KUKA KRL program: MyProgram_121().src

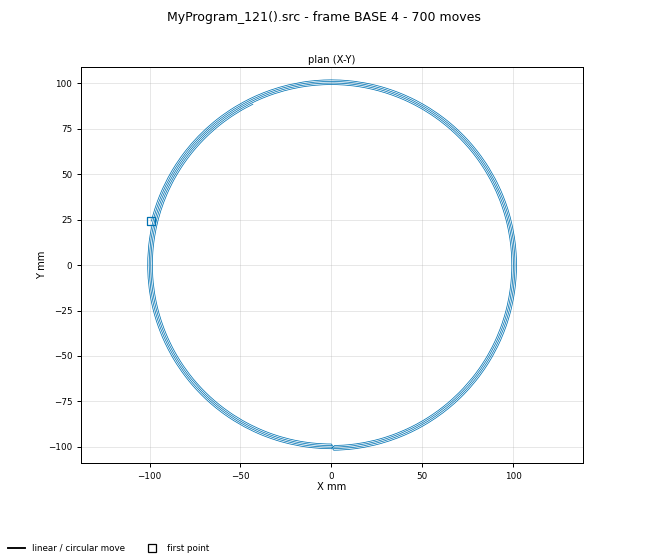
[picture p0: tool path of MyProgram_121().src in frame BASE 4, 700 of 700 moves have a stored position in this frame; points joined in program order, loops and branches not executed]
&ACCESS RVP
&REL 1
&PARAM TEMPLATE = C:\KRC\Roboter\Template\vorgabe
&PARAM EDITMASK = *
DEF MyProgram_121()
; ---- Setting reference (Base) ----
$BASE = BASE_DATA[4]

; --------------------------
; ---- Setting tool (TCP) ----
$TOOL = TOOL_DATA[3]
; --------------------------

$VEL.CP = VEL_APROX_PRINT
Startdeposition()
$VEL.CP = VEL_PRINT
LIN {X -98.957,Y 24.1948,Z 102,A 161.3136,B 24.9312,C -1.9162,E1 24.8447,E2 -75.7869} C_DIS
LIN {X -98.1679,Y 27.2258,Z 102,A 159.187,B 24.9317,C -1.9094,E1 24.8462,E2 -73.6317} C_DIS
LIN {X -97.1085,Y 30.7923,Z 102,A 156.6963,B 24.9321,C -1.9025,E1 24.8484,E2 -71.1104} C_DIS
LIN {X -95.7541,Y 34.7715,Z 102,A 155.0992,B 24.9297,C -1.9358,E1 24.8498,E2 -69.5835} C_DIS
LIN {X -94.7978,Y 37.2995,Z 102,A 153.5612,B 24.9294,C -1.9399,E1 24.8513,E2 -68.0466} C_DIS
LIN {X -93.6877,Y 40.0091,Z 102,A 151.9205,B 24.9291,C -1.9451,E1 24.8531,E2 -66.4092} C_DIS
LIN {X -92.7094,Y 42.2256,Z 102,A 150.3541,B 24.9293,C -1.9423,E1 24.8549,E2 -64.8275} C_DIS
LIN {X -89.881,Y 47.9536,Z 102,A 146.8815,B 24.9282,C -1.957,E1 24.8593,E2 -61.3714} C_DIS
LIN {X -87.5821,Y 52.0317,Z 102,A 144.2252,B 24.9277,C -1.9639,E1 24.8629,E2 -58.7175} C_DIS
LIN {X -85.5843,Y 55.2562,Z 102,A 141.634,B 24.9284,C -1.9543,E1 24.8668,E2 -56.0904} C_DIS
LIN {X -82.7794,Y 59.3759,Z 102,A 138.6498,B 24.9283,C -1.9558,E1 24.8717,E2 -53.0952} C_DIS
LIN {X -80.5027,Y 62.4283,Z 102,A 137.1356,B 24.9263,C -1.983,E1 24.8741,E2 -51.6386} C_DIS
LIN {X -76.9267,Y 66.7851,Z 102,A 134.0827,B 24.9254,C -1.9953,E1 24.8796,E2 -48.6009} C_DIS
LIN {X -73.2959,Y 70.7502,Z 102,A 130.9039,B 24.9252,C -1.9975,E1 24.8856,E2 -45.4133} C_DIS
LIN {X -69.1212,Y 74.8347,Z 102,A 127.7767,B 24.9242,C -2.0107,E1 24.8919,E2 -42.3047} C_DIS
LIN {X -64.7279,Y 78.6665,Z 102,A 124.3462,B 24.924,C -2.0128,E1 24.8991,E2 -38.8656} C_DIS
LIN {X -62.3244,Y 80.5828,Z 102,A 122.4933,B 24.924,C -2.0122,E1 24.9032,E2 -37.0044} C_DIS
LIN {X -60.1036,Y 82.2523,Z 102,A 120.9648,B 24.9237,C -2.0166,E1 24.9066,E2 -35.481} C_DIS
LIN {X -55.7725,Y 85.2492,Z 102,A 117.9876,B 24.9233,C -2.0219,E1 24.9135,E2 -32.5065} C_DIS
LIN {X -52.8849,Y 87.0693,Z 102,A 115.7015,B 24.924,C -2.0126,E1 24.919,E2 -30.1912} C_DIS
LIN {X -48.0016,Y 89.8555,Z 102,A 112.9772,B 24.9225,C -2.0335,E1 24.9255,E2 -27.5088} C_DIS
LIN {X -44.7125,Y 91.5369,Z 102,A 110.1519,B 24.9242,C -2.0105,E1 24.9327,E2 -24.6211} C_DIS
LIN {X -41.1942,Y 93.1711,Z 102,A 108.2639,B 24.9232,C -2.0241,E1 24.9375,E2 -22.761} C_DIS
LIN {X -37.1448,Y 94.8586,Z 102,A 106.1045,B 24.9221,C -2.0385,E1 24.943,E2 -20.631} C_DIS
LIN {X -33.5819,Y 96.1777,Z 102,A 103.6281,B 24.9228,C -2.0291,E1 24.9496,E2 -18.1274} C_DIS
LIN {X -28.5827,Y 97.7807,Z 102,A 101.0832,B 24.9214,C -2.0471,E1 24.9563,E2 -15.6207} C_DIS
LIN {X -23.5966,Y 99.1014,Z 102,A 97.8662,B 24.9221,C -2.0385,E1 24.965,E2 -12.3788} C_DIS
LIN {X -15.5786,Y 100.6736,Z 102,A 93.5985,B 24.9209,C -2.054,E1 24.9767,E2 -8.1433} C_DIS
LIN {X -12.7503,Y 101.0714,Z 102,A 91.1239,B 24.9232,C -2.0235,E1 24.9837,E2 -5.5944} C_DIS
LIN {X -8.267,Y 101.536,Z 102,A 89.0167,B 24.922,C -2.0402,E1 24.9895,E2 -3.5259} C_DIS
LIN {X -4.0963,Y 101.7898,Z 102,A 86.8934,B 24.9212,C -2.0493,E1 24.9953,E2 -1.4237} C_DIS
LIN {X -0.0604,Y 101.8734,Z 102,A 84.4498,B 24.9217,C -2.0434,E1 25.0022,E2 1.0339} C_DIS
LIN {X 4.8959,Y 101.7555,Z 102,A 81.9704,B 24.9208,C -2.0551,E1 25.009,E2 3.4849} C_DIS
LIN {X 8.4387,Y 101.5222,Z 102,A 79.9611,B 24.9208,C -2.0546,E1 25.0146,E2 5.4945} C_DIS
LIN {X 12.6527,Y 101.084,Z 102,A 77.4932,B 24.9211,C -2.051,E1 25.0215,E2 7.9692} C_DIS
LIN {X 18.3069,Y 100.2138,Z 102,A 74.5122,B 24.9205,C -2.0589,E1 25.0297,E2 10.9286} C_DIS
LIN {X 20.8892,Y 99.708,Z 102,A 72.5597,B 24.9219,C -2.0404,E1 25.0351,E2 12.9225} C_DIS
LIN {X 24.06,Y 98.9899,Z 102,A 70.5801,B 24.9224,C -2.0337,E1 25.0405,E2 14.9151} C_DIS
LIN {X 27.3534,Y 98.1318,Z 102,A 69.3081,B 24.9207,C -2.0567,E1 25.0438,E2 16.1306} C_DIS
LIN {X 29.7903,Y 97.4195,Z 102,A 67.1031,B 24.923,C -2.0262,E1 25.0499,E2 18.4039} C_DIS
LIN {X 33.4482,Y 96.2241,Z 102,A 65.5129,B 24.9215,C -2.0461,E1 25.0539,E2 19.9437} C_DIS
LIN {X 36.8556,Y 94.9721,Z 102,A 63.4452,B 24.9217,C -2.0432,E1 25.0593,E2 22.014} C_DIS
LIN {X 39.9474,Y 93.7137,Z 102,A 60.8845,B 24.9239,C -2.0151,E1 25.0661,E2 24.6351} C_DIS
LIN {X 43.9838,Y 91.8875,Z 102,A 59.4721,B 24.9209,C -2.0535,E1 25.0694,E2 25.9529} C_DIS
LIN {X 46.2574,Y 90.7642,Z 102,A 56.8281,B 24.9246,C -2.0049,E1 25.0763,E2 28.7047} C_DIS
LIN {X 50.6903,Y 88.365,Z 102,A 54.8585,B 24.9224,C -2.0341,E1 25.0809,E2 30.5994} C_DIS
LIN {X 54.1717,Y 86.2749,Z 102,A 52.6742,B 24.9224,C -2.0345,E1 25.0861,E2 32.7759} C_DIS
LIN {X 58.6838,Y 83.2733,Z 102,A 49.6805,B 24.9226,C -2.0316,E1 25.093,E2 35.7664} C_DIS
LIN {X 62.2919,Y 80.6078,Z 102,A 46.5734,B 24.9247,C -2.0044,E1 25.1,E2 38.9267} C_DIS
LIN {X 65.02,Y 78.4237,Z 102,A 45.1697,B 24.9233,C -2.0226,E1 25.103,E2 40.2819} C_DIS
LIN {X 67.3026,Y 76.4747,Z 102,A 43.2946,B 24.9241,C -2.0119,E1 25.1069,E2 42.1748} C_DIS
LIN {X 70.2619,Y 73.7665,Z 102,A 41.0725,B 24.9243,C -2.0086,E1 25.1115,E2 44.3956} C_DIS
LIN {X 72.8301,Y 71.2314,Z 102,A 38.6497,B 24.9258,C -1.9888,E1 25.1163,E2 46.8551} C_DIS
LIN {X 75.2471,Y 68.6719,Z 102,A 37.241,B 24.9245,C -2.007,E1 25.1189,E2 48.2146} C_DIS
LIN {X 77.6522,Y 65.9396,Z 102,A 35.1787,B 24.9249,C -2.0017,E1 25.1227,E2 50.2801} C_DIS
LIN {X 80.2578,Y 62.7425,Z 102,A 32.7459,B 24.9256,C -1.9916,E1 25.1269,E2 52.7253} C_DIS
LIN {X 82.4053,Y 59.8946,Z 102,A 30.0003,B 24.9282,C -1.9573,E1 25.1316,E2 55.5388} C_DIS
LIN {X 85.1755,Y 55.8844,Z 102,A 28.2311,B 24.9258,C -1.9889,E1 25.1342,E2 57.2245} C_DIS
LIN {X 86.6688,Y 53.541,Z 102,A 26.463,B 24.9267,C -1.9766,E1 25.1368,E2 59.0128} C_DIS
LIN {X 90.1368,Y 47.4683,Z 102,A 23.0663,B 24.9259,C -1.9876,E1 25.1414,E2 62.3659} C_DIS
LIN {X 91.2122,Y 45.3677,Z 102,A 20.6112,B 24.9296,C -1.9384,E1 25.1446,E2 64.9238} C_DIS
LIN {X 93.1278,Y 41.2972,Z 102,A 18.7221,B 24.9282,C -1.9569,E1 25.1467,E2 66.7591} C_DIS
LIN {X 94.3777,Y 38.3499,Z 102,A 17.0093,B 24.9283,C -1.9553,E1 25.1486,E2 68.4663} C_DIS
LIN {X 95.8893,Y 34.397,Z 102,A 14.3971,B 24.9295,C -1.9389,E1 25.1511,E2 71.1026} C_DIS
LIN {X 97.1898,Y 30.5313,Z 102,A 11.7186,B 24.9311,C -1.9164,E1 25.1534,E2 73.8189} C_DIS
LIN {X 98.3574,Y 26.5274,Z 102,A 10.298,B 24.9289,C -1.9468,E1 25.1544,E2 75.1597} C_DIS
LIN {X 99.6077,Y 21.3614,Z 102,A 6.9761,B 24.9306,C -1.9239,E1 25.1566,E2 78.5162} C_DIS
LIN {X 100.689,Y 15.4791,Z 102,A 3.8424,B 24.9306,C -1.9228,E1 25.1581,E2 81.6344} C_DIS
LIN {X 101.1414,Y 12.1818,Z 102,A 1.9937,B 24.9311,C -1.9177,E1 25.1587,E2 83.484} C_DIS
LIN {X 101.4335,Y 9.4408,Z 102,A 0.3861,B 24.9316,C -1.9105,E1 25.1592,E2 85.0993} C_DIS
LIN {X 101.674,Y 6.3658,Z 102,A -1.3493,B 24.932,C -1.9049,E1 25.1595,E2 86.8376} C_DIS
LIN {X 101.8206,Y 3.2332,Z 102,A -3.1874,B 24.9326,C -1.8962,E1 25.1597,E2 88.6853} C_DIS
LIN {X 101.8681,Y -0.9186,Z 102,A -5.3811,B 24.9327,C -1.8944,E1 25.1597,E2 90.87} C_DIS
LIN {X 101.8011,Y -3.8335,Z 102,A -7.1036,B 24.9333,C -1.8857,E1 25.1597,E2 92.6028} C_DIS
LIN {X 101.583,Y -7.6782,Z 102,A -9.614,B 24.9348,C -1.8646,E1 25.1591,E2 95.148} C_DIS
LIN {X 101.202,Y -11.6643,Z 102,A -11.454,B 24.9342,C -1.8742,E1 25.1586,E2 96.9545} C_DIS
LIN {X 100.7976,Y -14.7613,Z 102,A -13.7844,B 24.9362,C -1.8451,E1 25.1577,E2 99.3398} C_DIS
LIN {X 100.1615,Y -18.5978,Z 102,A -15.2787,B 24.9347,C -1.8663,E1 25.157,E2 100.7753} C_DIS
LIN {X 98.9392,Y -24.2676,Z 102,A -18.5433,B 24.9354,C -1.8558,E1 25.155,E2 104.0458} C_DIS
LIN {X 98.1116,Y -27.4247,Z 102,A -21.1732,B 24.9381,C -1.8176,E1 25.153,E2 106.7506} C_DIS
LIN {X 96.8209,Y -31.6811,Z 102,A -22.8366,B 24.9363,C -1.8439,E1 25.1516,E2 108.3428} C_DIS
LIN {X 96.1216,Y -33.7417,Z 102,A -24.1234,B 24.9367,C -1.8375,E1 25.1504,E2 109.6374} C_DIS
LIN {X 94.8323,Y -37.2115,Z 102,A -26.9146,B 24.9391,C -1.8022,E1 25.1475,E2 112.4963} C_DIS
LIN {X 93.1267,Y -41.2996,Z 102,A -28.5864,B 24.9374,C -1.8279,E1 25.1458,E2 114.0984} C_DIS
LIN {X 91.508,Y -44.771,Z 102,A -30.9615,B 24.9384,C -1.8124,E1 25.1429,E2 116.4973} C_DIS
LIN {X 88.6903,Y -50.1215,Z 102,A -34.4418,B 24.9393,C -1.7991,E1 25.1382,E2 119.9906} C_DIS
LIN {X 86.7386,Y -53.4291,Z 102,A -36.3016,B 24.9389,C -1.8051,E1 25.1356,E2 121.8267} C_DIS
LIN {X 84.2579,Y -57.2583,Z 102,A -38.9024,B 24.9395,C -1.7965,E1 25.1316,E2 124.435} C_DIS
LIN {X 81.5429,Y -61.0626,Z 102,A -41.5712,B 24.9401,C -1.7876,E1 25.1272,E2 127.1117} C_DIS
LIN {X 79.8337,Y -63.2809,Z 102,A -43.2837,B 24.9408,C -1.7778,E1 25.1242,E2 128.8393} C_DIS
LIN {X 75.9735,Y -67.8669,Z 102,A -47.1166,B 24.9426,C -1.7506,E1 25.1171,E2 132.7191} C_DIS
LIN {X 73.0436,Y -71.0119,Z 102,A -48.7286,B 24.9408,C -1.7769,E1 25.1141,E2 134.2621} C_DIS
LIN {X 71.0205,Y -73.0344,Z 102,A -51.1432,B 24.9432,C -1.7407,E1 25.1092,E2 136.752} C_DIS
LIN {X 67.8525,Y -75.9864,Z 102,A -53.4227,B 24.9432,C -1.7413,E1 25.1044,E2 139.0211} C_DIS
LIN {X 64.9851,Y -78.4528,Z 102,A -54.9479,B 24.9419,C -1.7605,E1 25.1013,E2 140.4949} C_DIS
LIN {X 61.2987,Y -81.3656,Z 102,A -57.8925,B 24.9431,C -1.7428,E1 25.0947,E2 143.4707} C_DIS
LIN {X 57.2695,Y -84.2503,Z 102,A -60.716,B 24.9435,C -1.7356,E1 25.0882,E2 146.3013} C_DIS
LIN {X 53.6209,Y -86.619,Z 102,A -62.9616,B 24.9433,C -1.7389,E1 25.083,E2 148.532} C_DIS
LIN {X 49.9889,Y -88.7644,Z 102,A -65.0648,B 24.9429,C -1.7453,E1 25.0779,E2 150.6137} C_DIS
LIN {X 47.3229,Y -90.2133,Z 102,A -67.4241,B 24.9448,C -1.7166,E1 25.072,E2 153.0342} C_DIS
LIN {X 44.023,Y -91.8687,Z 102,A -68.4874,B 24.9424,C -1.7532,E1 25.0695,E2 154.0081} C_DIS
LIN {X 40.1747,Y -93.6173,Z 102,A -71.5204,B 24.9443,C -1.7236,E1 25.0616,E2 157.1036} C_DIS
LIN {X 36.6974,Y -95.0343,Z 102,A -73.318,B 24.9437,C -1.733,E1 25.057,E2 158.875} C_DIS
LIN {X 31.9978,Y -96.7166,Z 102,A -76.5016,B 24.9449,C -1.7147,E1 25.0485,E2 162.0955} C_DIS
LIN {X 27.2491,Y -98.1614,Z 102,A -79.0163,B 24.9444,C -1.7223,E1 25.0419,E2 164.5878} C_DIS
LIN {X 24.1297,Y -98.9729,Z 102,A -80.818,B 24.9444,C -1.7209,E1 25.037,E2 166.3901} C_DIS
LIN {X 18.0332,Y -100.263,Z 102,A -84.1356,B 24.9442,C -1.7251,E1 25.028,E2 169.6937} C_DIS
LIN {X 13.4852,Y -100.9761,Z 102,A -86.6996,B 24.9442,C -1.7242,E1 25.0209,E2 172.2575} C_DIS
LIN {X 9.4028,Y -101.437,Z 102,A -89.149,B 24.9447,C -1.7175,E1 25.014,E2 174.721} C_DIS
LIN {X 3.7497,Y -101.8047,Z 102,A -92.3082,B 24.9447,C -1.7172,E1 25.0052,E2 177.8798} C_DIS
LIN {X 1.335,Y -101.8645,Z 102,A -93.9063,B 24.9454,C -1.7077,E1 25.0007,E2 179.5002} C_DIS
LIN {X 1.335,Y -101.8645,Z 102,A -93.9063,B 24.9454,C -1.7077,E1 25.0007,E2 179.5002} C_DIS
Enddeposition()
LIN {X 0.7041,Y -101.0045,Z 102,A -93.5064,B 24.9425,C -1.7514,E1 25.0021,E2 178.9966} C_DIS
Startdeposition()
$VEL.CP = VEL_PRINT
LIN {X 3.718,Y -100.9431,Z 102,A -91.511,B 24.9418,C -1.7629,E1 25.0078,E2 176.9745} C_DIS
LIN {X 9.5388,Y -100.5585,Z 102,A -88.2058,B 24.9417,C -1.7643,E1 25.017,E2 173.6676} C_DIS
LIN {X 12.8674,Y -100.1867,Z 102,A -85.5674,B 24.9397,C -1.7943,E1 25.0245,E2 170.9602} C_DIS
LIN {X 17.6276,Y -99.4599,Z 102,A -83.9549,B 24.9424,C -1.7527,E1 25.0286,E2 169.4478} C_DIS
LIN {X 24.2532,Y -98.0552,Z 102,A -79.9432,B 24.9418,C -1.7627,E1 25.0396,E2 165.4177} C_DIS
LIN {X 29.2648,Y -96.679,Z 102,A -77.062,B 24.9418,C -1.7632,E1 25.0474,E2 162.5399} C_DIS
LIN {X 32.894,Y -95.5051,Z 102,A -74.7112,B 24.9411,C -1.7732,E1 25.0536,E2 160.1701} C_DIS
LIN {X 35.8349,Y -94.4394,Z 102,A -73.0166,B 24.9411,C -1.7725,E1 25.0581,E2 158.4807} C_DIS
LIN {X 39.1276,Y -93.1235,Z 102,A -70.5763,B 24.9398,C -1.7924,E1 25.0645,E2 155.999} C_DIS
LIN {X 42.0663,Y -91.8354,Z 102,A -69.1318,B 24.9406,C -1.7803,E1 25.0681,E2 154.5869} C_DIS
LIN {X 44.7528,Y -90.5546,Z 102,A -66.8651,B 24.9389,C -1.8061,E1 25.0739,E2 152.265} C_DIS
LIN {X 48.2344,Y -88.749,Z 102,A -65.0382,B 24.9397,C -1.794,E1 25.0783,E2 150.4719} C_DIS
LIN {X 53.0415,Y -85.9642,Z 102,A -62.0296,B 24.9397,C -1.7941,E1 25.0855,E2 147.4725} C_DIS
LIN {X 55.7068,Y -84.2598,Z 102,A -60.1387,B 24.9392,C -1.8015,E1 25.0899,E2 145.5703} C_DIS
LIN {X 58.4209,Y -82.4016,Z 102,A -58.5337,B 24.9396,C -1.7948,E1 25.0935,E2 143.9866} C_DIS
LIN {X 62.8557,Y -79.0707,Z 102,A -55.2313,B 24.9387,C -1.8078,E1 25.1009,E2 140.6655} C_DIS
LIN {X 65.2536,Y -77.1039,Z 102,A -53.2996,B 24.938,C -1.8188,E1 25.1051,E2 138.7154} C_DIS
LIN {X 69.5185,Y -73.2813,Z 102,A -50.021,B 24.9374,C -1.8276,E1 25.1118,E2 135.4292} C_DIS
LIN {X 72.6836,Y -70.1429,Z 102,A -48.0689,B 24.9386,C -1.8105,E1 25.1156,E2 133.526} C_DIS
LIN {X 75.3334,Y -67.2892,Z 102,A -45.4026,B 24.9369,C -1.8346,E1 25.1207,E2 130.8144} C_DIS
LIN {X 79.0683,Y -62.8588,Z 102,A -42.3682,B 24.937,C -1.833,E1 25.126,E2 127.7979} C_DIS
LIN {X 81.8233,Y -59.2299,Z 102,A -39.6853,B 24.9363,C -1.844,E1 25.1305,E2 125.1019} C_DIS
LIN {X 84.2139,Y -55.7763,Z 102,A -37.3625,B 24.936,C -1.8482,E1 25.1342,E2 122.7805} C_DIS
LIN {X 86.0318,Y -52.9318,Z 102,A -35.1793,B 24.9348,C -1.8647,E1 25.1374,E2 120.5695} C_DIS
LIN {X 87.8918,Y -49.7829,Z 102,A -33.0178,B 24.9341,C -1.8743,E1 25.1404,E2 118.3964} C_DIS
LIN {X 89.4405,Y -46.94,Z 102,A -31.1164,B 24.9336,C -1.8825,E1 25.1429,E2 116.4859} C_DIS
LIN {X 91.0724,Y -43.6895,Z 102,A -29.9725,B 24.9358,C -1.8509,E1 25.1442,E2 115.4227} C_DIS
LIN {X 92.7456,Y -40.0134,Z 102,A -27.118,B 24.9337,C -1.8809,E1 25.1475,E2 112.5129} C_DIS
LIN {X 94.7381,Y -35.0406,Z 102,A -24.2575,B 24.9335,C -1.8829,E1 25.1504,E2 109.6635} C_DIS
LIN {X 95.7786,Y -32.085,Z 102,A -22.0553,B 24.9319,C -1.9061,E1 25.1524,E2 107.4192} C_DIS
LIN {X 96.816,Y -28.8028,Z 102,A -20.1106,B 24.9315,C -1.9119,E1 25.154,E2 105.4717} C_DIS
LIN {X 97.7554,Y -25.4345,Z 102,A -18.5556,B 24.9323,C -1.9005,E1 25.155,E2 103.9527} C_DIS
LIN {X 99.2082,Y -18.9919,Z 102,A -13.9565,B 24.9289,C -1.9479,E1 25.1577,E2 99.2686} C_DIS
LIN {X 100.0692,Y -13.7587,Z 102,A -11.8356,B 24.9308,C -1.9206,E1 25.1585,E2 97.2244} C_DIS
LIN {X 100.5142,Y -9.9945,Z 102,A -9.5934,B 24.9301,C -1.9314,E1 25.1592,E2 94.97} C_DIS
LIN {X 100.8057,Y -6.4192,Z 102,A -7.7095,B 24.9301,C -1.9318,E1 25.1595,E2 93.0965} C_DIS
LIN {X 100.9662,Y -2.9641,Z 102,A -5.8376,B 24.9298,C -1.9344,E1 25.1597,E2 91.2295} C_DIS
LIN {X 101.0094,Y 0.3369,Z 102,A -3.8497,B 24.9291,C -1.9452,E1 25.1597,E2 89.228} C_DIS
LIN {X 100.919,Y 4.2775,Z 102,A -1.7641,B 24.929,C -1.9462,E1 25.1596,E2 87.1524} C_DIS
LIN {X 100.7363,Y 7.45,Z 102,A 0.1445,B 24.9282,C -1.9563,E1 25.1592,E2 85.2313} C_DIS
LIN {X 100.4092,Y 11.008,Z 102,A 1.982,B 24.9283,C -1.955,E1 25.1587,E2 83.4077} C_DIS
LIN {X 99.9242,Y 14.7796,Z 102,A 4.0607,B 24.9281,C -1.9586,E1 25.1579,E2 81.3327} C_DIS
LIN {X 98.8915,Y 20.5788,Z 102,A 7.3682,B 24.9274,C -1.9677,E1 25.1563,E2 78.0233} C_DIS
LIN {X 97.5641,Y 26.1578,Z 102,A 11.2889,B 24.9246,C -2.0051,E1 25.1536,E2 74.037} C_DIS
LIN {X 96.5587,Y 29.6552,Z 102,A 12.7772,B 24.9259,C -1.9877,E1 25.1524,E2 72.5983} C_DIS
LIN {X 95.6449,Y 32.4813,Z 102,A 15.0609,B 24.9237,C -2.0173,E1 25.1503,E2 70.2576} C_DIS
LIN {X 94.3461,Y 36.0813,Z 102,A 16.6989,B 24.9249,C -2.0018,E1 25.1488,E2 68.6652} C_DIS
LIN {X 93.1086,Y 39.1628,Z 102,A 18.4759,B 24.9248,C -2.0029,E1 25.1469,E2 66.8954} C_DIS
LIN {X 90.1455,Y 45.5733,Z 102,A 22.3155,B 24.9244,C -2.0074,E1 25.1423,E2 63.0657} C_DIS
LIN {X 86.9566,Y 51.3954,Z 102,A 26.222,B 24.9232,C -2.0233,E1 25.137,E2 59.1422} C_DIS
LIN {X 85.1122,Y 54.3958,Z 102,A 28.1843,B 24.9229,C -2.0271,E1 25.1341,E2 57.1808} C_DIS
LIN {X 82.2818,Y 58.5889,Z 102,A 31.1035,B 24.9222,C -2.0364,E1 25.1295,E2 54.254} C_DIS
LIN {X 80.0842,Y 61.5587,Z 102,A 33.6852,B 24.9203,C -2.0611,E1 25.125,E2 51.6263} C_DIS
LIN {X 77.8382,Y 64.3756,Z 102,A 35.2747,B 24.9214,C -2.0477,E1 25.1223,E2 50.0759} C_DIS
LIN {X 75.6284,Y 66.9596,Z 102,A 37.7089,B 24.9195,C -2.0724,E1 25.1177,E2 47.5943} C_DIS
LIN {X 73.0313,Y 69.7823,Z 102,A 39.3544,B 24.9207,C -2.0559,E1 25.1146,E2 45.9949} C_DIS
LIN {X 70.5312,Y 72.3094,Z 102,A 41.3938,B 24.9203,C -2.0611,E1 25.1106,E2 43.9518} C_DIS
LIN {X 68.6184,Y 74.126,Z 102,A 42.8116,B 24.9203,C -2.0611,E1 25.1077,E2 42.5398} C_DIS
LIN {X 66.2967,Y 76.2084,Z 102,A 44.6256,B 24.9199,C -2.0663,E1 25.1039,E2 40.7206} C_DIS
LIN {X 64.2384,Y 77.9522,Z 102,A 46.9478,B 24.9172,C -2.1007,E1 25.0987,E2 38.3258} C_DIS
LIN {X 60.3069,Y 81.0322,Z 102,A 48.9663,B 24.9194,C -2.0734,E1 25.0944,E2 36.3792} C_DIS
LIN {X 57.4956,Y 83.0496,Z 102,A 51.2413,B 24.9182,C -2.089,E1 25.0891,E2 34.0751} C_DIS
LIN {X 53.9627,Y 85.3888,Z 102,A 53.3987,B 24.9186,C -2.0831,E1 25.0841,E2 31.9388} C_DIS
LIN {X 50.6347,Y 87.4025,Z 102,A 55.3916,B 24.919,C -2.078,E1 25.0793,E2 29.964} C_DIS
LIN {X 44.6462,Y 90.6075,Z 102,A 59.0891,B 24.919,C -2.077,E1 25.0703,E2 26.2793} C_DIS
LIN {X 39.6203,Y 92.9159,Z 102,A 62.4898,B 24.918,C -2.0908,E1 25.0615,E2 22.8545} C_DIS
LIN {X 36.2101,Y 94.2973,Z 102,A 64.49,B 24.9181,C -2.0895,E1 25.0563,E2 20.8618} C_DIS
LIN {X 30.4974,Y 96.2971,Z 102,A 68.0603,B 24.9175,C -2.0976,E1 25.0469,E2 17.2792} C_DIS
LIN {X 27.0963,Y 97.3085,Z 102,A 69.8783,B 24.918,C -2.0916,E1 25.042,E2 15.4786} C_DIS
LIN {X 23.1525,Y 98.3213,Z 102,A 73.0181,B 24.9153,C -2.1247,E1 25.0333,E2 12.2649} C_DIS
LIN {X 18.6591,Y 99.2722,Z 102,A 74.6164,B 24.9183,C -2.0874,E1 25.0292,E2 10.7568} C_DIS
LIN {X 13.649,Y 100.0848,Z 102,A 77.6208,B 24.9178,C -2.093,E1 25.0209,E2 7.7422} C_DIS
LIN {X 9.0501,Y 100.6036,Z 102,A 80.314,B 24.9176,C -2.0959,E1 25.0134,E2 5.0438} C_DIS
LIN {X 5.5342,Y 100.8579,Z 102,A 82.8155,B 24.9161,C -2.1148,E1 25.0063,E2 2.4986} C_DIS
LIN {X 2.1141,Y 100.9878,Z 102,A 84.7803,B 24.9161,C -2.1154,E1 25.0008,E2 0.5326} C_DIS
LIN {X -1.4149,Y 101.0007,Z 102,A 86.2851,B 24.9176,C -2.0964,E1 24.9967,E2 -0.927} C_DIS
LIN {X -4.1801,Y 100.9232,Z 102,A 87.6033,B 24.9183,C -2.0866,E1 24.9931,E2 -2.2224} C_DIS
LIN {X -8.8933,Y 100.6181,Z 102,A 90.8211,B 24.9169,C -2.1053,E1 24.984,E2 -5.4858} C_DIS
LIN {X -14.9513,Y 99.8981,Z 102,A 95.308,B 24.914,C -2.1413,E1 24.9714,E2 -10.0618} C_DIS
LIN {X -21.3961,Y 98.7176,Z 102,A 97.3834,B 24.919,C -2.0777,E1 24.9661,E2 -11.9885} C_DIS
LIN {X -26.7721,Y 97.3981,Z 102,A 100.9042,B 24.9182,C -2.0884,E1 24.9565,E2 -15.5397} C_DIS
LIN {X -29.9761,Y 96.4592,Z 102,A 103.0901,B 24.9175,C -2.0969,E1 24.9506,E2 -17.7495} C_DIS
LIN {X -34.3267,Y 94.9985,Z 102,A 105.482,B 24.9184,C -2.086,E1 24.9443,E2 -20.1201} C_DIS
LIN {X -37.6329,Y 93.7387,Z 102,A 108.495,B 24.9157,C -2.1197,E1 24.9363,E2 -23.22} C_DIS
LIN {X -42.9207,Y 91.4378,Z 102,A 110.7457,B 24.919,C -2.0778,E1 24.9308,E2 -25.3765} C_DIS
LIN {X -45.7655,Y 90.0473,Z 102,A 112.4606,B 24.9195,C -2.072,E1 24.9266,E2 -27.0822} C_DIS
LIN {X -48.1872,Y 88.7746,Z 102,A 114.1902,B 24.9192,C -2.0757,E1 24.9223,E2 -28.8255} C_DIS
LIN {X -53.362,Y 85.7641,Z 102,A 117.4807,B 24.92,C -2.0657,E1 24.9144,E2 -32.1023} C_DIS
LIN {X -56.8836,Y 83.4698,Z 102,A 120.2515,B 24.9193,C -2.0748,E1 24.9079,E2 -34.9039} C_DIS
LIN {X -61.2491,Y 80.3228,Z 102,A 123.0969,B 24.9203,C -2.0611,E1 24.9016,E2 -37.7268} C_DIS
LIN {X -64.1777,Y 78.0026,Z 102,A 125.8487,B 24.919,C -2.0788,E1 24.8955,E2 -40.5313} C_DIS
LIN {X -67.7132,Y 74.9538,Z 102,A 127.8059,B 24.9213,C -2.0484,E1 24.8916,E2 -42.4236} C_DIS
LIN {X -71.8163,Y 71.0308,Z 102,A 130.882,B 24.9223,C -2.0356,E1 24.8855,E2 -45.4823} C_DIS
LIN {X -75.4985,Y 67.1047,Z 102,A 134.1162,B 24.9224,C -2.0343,E1 24.8793,E2 -48.7274} C_DIS
LIN {X -77.2055,Y 65.1344,Z 102,A 135.9263,B 24.9218,C -2.042,E1 24.876,E2 -50.5642} C_DIS
LIN {X -79.8575,Y 61.8529,Z 102,A 138.2332,B 24.9225,C -2.0326,E1 24.8721,E2 -52.8596} C_DIS
LIN {X -83.1756,Y 57.3143,Z 102,A 142.0046,B 24.9216,C -2.0442,E1 24.866,E2 -56.6772} C_DIS
LIN {X -85.9099,Y 53.1285,Z 102,A 144.0865,B 24.9243,C -2.0099,E1 24.863,E2 -58.6878} C_DIS
LIN {X -88.3186,Y 49.0187,Z 102,A 146.9225,B 24.9245,C -2.0067,E1 24.859,E2 -61.531} C_DIS
LIN {X -91.0372,Y 43.7627,Z 102,A 149.9872,B 24.926,C -1.9867,E1 24.8552,E2 -64.5645} C_DIS
LIN {X -92.1723,Y 41.3188,Z 102,A 151.6058,B 24.9261,C -1.9851,E1 24.8533,E2 -66.1882} C_DIS
LIN {X -93.3631,Y 38.5557,Z 102,A 153.4343,B 24.9261,C -1.9841,E1 24.8513,E2 -68.0244} C_DIS
LIN {X -94.8874,Y 34.6314,Z 102,A 156.2752,B 24.9256,C -1.9923,E1 24.8485,E2 -70.9011} C_DIS
LIN {X -96.0871,Y 31.1484,Z 102,A 157.7366,B 24.9277,C -1.9642,E1 24.8473,E2 -72.3037} C_DIS
LIN {X -97.1774,Y 27.559,Z 102,A 159.91,B 24.928,C -1.9591,E1 24.8456,E2 -74.4774} C_DIS
LIN {X -97.885,Y 24.9301,Z 102,A 161.4707,B 24.9284,C -1.9547,E1 24.8445,E2 -76.0368} C_DIS
LIN {X -98.888,Y 20.5959,Z 102,A 163.8033,B 24.9294,C -1.9402,E1 24.8431,E2 -78.3484} C_DIS
LIN {X -99.6185,Y 16.7062,Z 102,A 166.3138,B 24.9293,C -1.942,E1 24.8418,E2 -80.8781} C_DIS
LIN {X -100.1041,Y 13.5055,Z 102,A 168.2412,B 24.9295,C -1.9392,E1 24.841,E2 -82.8104} C_DIS
LIN {X -100.4319,Y 10.7913,Z 102,A 170.0378,B 24.9292,C -1.9426,E1 24.8405,E2 -84.6259} C_DIS
LIN {X -100.9418,Y 3.7475,Z 102,A 173.6667,B 24.9311,C -1.9167,E1 24.8399,E2 -88.2149} C_DIS
LIN {X -100.991,Y -1.9409,Z 102,A 176.9167,B 24.9318,C -1.9071,E1 24.8399,E2 -91.4614} C_DIS
LIN {X -100.7524,Y -7.2157,Z 102,A 179.8213,B 24.9327,C -1.8944,E1 24.8403,E2 -94.3532} C_DIS
LIN {X -100.1563,Y -13.1027,Z 102,A -176.9739,B 24.9339,C -1.8785,E1 24.8412,E2 -97.5392} C_DIS
LIN {X -99.5167,Y -17.312,Z 102,A -174.0962,B 24.9333,C -1.8866,E1 24.8424,E2 -100.4535} C_DIS
LIN {X -98.8978,Y -20.548,Z 102,A -172.507,B 24.9344,C -1.8712,E1 24.8433,E2 -102.0153} C_DIS
LIN {X -98.0592,Y -24.237,Z 102,A -170.1101,B 24.9342,C -1.8732,E1 24.8448,E2 -104.431} C_DIS
LIN {X -97.2197,Y -27.4097,Z 102,A -168.1983,B 24.9345,C -1.8693,E1 24.8462,E2 -106.3446} C_DIS
LIN {X -96.2722,Y -30.5761,Z 102,A -166.2901,B 24.9348,C -1.8647,E1 24.8478,E2 -108.253} C_DIS
LIN {X -95.1679,Y -33.8556,Z 102,A -164.2587,B 24.9351,C -1.8613,E1 24.8497,E2 -110.2876} C_DIS
LIN {X -93.9248,Y -37.1636,Z 102,A -162.2855,B 24.9355,C -1.8543,E1 24.8516,E2 -112.2554} C_DIS
LIN {X -92.7858,Y -39.9246,Z 102,A -160.1546,B 24.9348,C -1.8647,E1 24.854,E2 -114.4227} C_DIS
LIN {X -91.3647,Y -43.0775,Z 102,A -158.5821,B 24.9362,C -1.8455,E1 24.8558,E2 -115.9581} C_DIS
LIN {X -89.8469,Y -46.1575,Z 102,A -156.5837,B 24.9364,C -1.8419,E1 24.8584,E2 -117.9586} C_DIS
LIN {X -87.9053,Y -49.7589,Z 102,A -154.2557,B 24.9368,C -1.8358,E1 24.8615,E2 -120.2843} C_DIS
LIN {X -86.3208,Y -52.4562,Z 102,A -152.6141,B 24.9375,C -1.8265,E1 24.8638,E2 -121.9122} C_DIS
LIN {X -84.9967,Y -54.5756,Z 102,A -150.8282,B 24.9368,C -1.8358,E1 24.8666,E2 -123.7292} C_DIS
LIN {X -82.2719,Y -58.6027,Z 102,A -148.3866,B 24.9381,C -1.8177,E1 24.8704,E2 -126.1397} C_DIS
LIN {X -80.201,Y -61.4071,Z 102,A -146.3824,B 24.9383,C -1.8138,E1 24.8738,E2 -128.1442} C_DIS
LIN {X -78.2074,Y -63.9275,Z 102,A -144.6163,B 24.9388,C -1.8074,E1 24.8768,E2 -129.9035} C_DIS
LIN {X -76.2576,Y -66.2405,Z 102,A -142.3471,B 24.9377,C -1.8232,E1 24.8811,E2 -132.2205} C_DIS
LIN {X -73.9516,Y -68.8042,Z 102,A -140.8777,B 24.9392,C -1.8015,E1 24.8838,E2 -133.6447} C_DIS
LIN {X -71.6605,Y -71.1885,Z 102,A -138.892,B 24.9392,C -1.8014,E1 24.8877,E2 -135.6387} C_DIS
LIN {X -69.0195,Y -73.7517,Z 102,A -136.9111,B 24.9397,C -1.7933,E1 24.8917,E2 -137.6084} C_DIS
LIN {X -66.8631,Y -75.7138,Z 102,A -134.5316,B 24.9382,C -1.8161,E1 24.8968,E2 -140.0517} C_DIS
LIN {X -63.6431,Y -78.4379,Z 102,A -132.8231,B 24.9402,C -1.787,E1 24.9003,E2 -141.6972} C_DIS
LIN {X -60.8702,Y -80.6091,Z 102,A -130.841,B 24.9404,C -1.7828,E1 24.9047,E2 -143.6767} C_DIS
LIN {X -58.9528,Y -82.0218,Z 102,A -129.3662,B 24.9403,C -1.785,E1 24.9081,E2 -145.1618} C_DIS
LIN {X -56.5912,Y -83.6683,Z 102,A -127.8395,B 24.9407,C -1.7785,E1 24.9116,E2 -146.6782} C_DIS
LIN {X -53.6179,Y -85.6042,Z 102,A -125.8401,B 24.941,C -1.7749,E1 24.9163,E2 -148.6755} C_DIS
LIN {X -47.8269,Y -88.9701,Z 102,A -121.948,B 24.941,C -1.7729,E1 24.9257,E2 -152.5743} C_DIS
LIN {X -42.6424,Y -91.5673,Z 102,A -118.8686,B 24.9419,C -1.7612,E1 24.9334,E2 -155.6339} C_DIS
LIN {X -39.5835,Y -92.9313,Z 102,A -116.7499,B 24.9415,C -1.7671,E1 24.9388,E2 -157.7718} C_DIS
LIN {X -37.2719,Y -93.8823,Z 102,A -114.6446,B 24.9399,C -1.7913,E1 24.9445,E2 -159.9391} C_DIS
LIN {X -33.1469,Y -95.4166,Z 102,A -112.7806,B 24.9416,C -1.7656,E1 24.9492,E2 -161.7456} C_DIS
LIN {X -29.8579,Y -96.4959,Z 102,A -110.9668,B 24.942,C -1.7585,E1 24.954,E2 -163.5458} C_DIS
LIN {X -27.455,Y -97.2068,Z 102,A -109.5634,B 24.9422,C -1.7569,E1 24.9578,E2 -164.9477} C_DIS
LIN {X -23.1067,Y -98.3319,Z 102,A -106.9409,B 24.9421,C -1.7582,E1 24.9649,E2 -167.5771} C_DIS
LIN {X -16.7717,Y -99.6075,Z 102,A -103.5225,B 24.9428,C -1.7475,E1 24.9742,E2 -170.9738} C_DIS
LIN {X -13.9343,Y -100.0443,Z 102,A -101.6061,B 24.9421,C -1.7579,E1 24.9796,E2 -172.9166} C_DIS
LIN {X -10.2953,Y -100.4838,Z 102,A -99.4391,B 24.9419,C -1.761,E1 24.9856,E2 -175.0922} C_DIS
LIN {X -6.5219,Y -100.7993,Z 102,A -97.3766,B 24.9421,C -1.7577,E1 24.9913,E2 -177.1477} C_DIS
LIN {X -2.9848,Y -100.9656,Z 102,A -95.4563,B 24.9423,C -1.7546,E1 24.9967,E2 -179.061} C_DIS
LIN {X 0.1794,Y -101.0104,Z 102,A -93.5269,B 24.9419,C -1.7601,E1 25.0021,E2 -181.0034} C_DIS
LIN {X 0.1794,Y -101.0104,Z 102,A -93.5269,B 24.9419,C -1.7601,E1 25.0021,E2 -181.0034} C_DIS
Enddeposition()
LIN {X 0.6945,Y -100.1423,Z 102,A -93.5343,B 24.9417,C -1.7637,E1 25.0021,E2 -181.0047} C_DIS
Startdeposition()
$VEL.CP = VEL_PRINT
LIN {X -1.645,Y -100.1341,Z 102,A -95.5352,B 24.9434,C -1.7386,E1 24.9964,E2 -178.9441} C_DIS
LIN {X -4.8806,Y -100.0301,Z 102,A -97.4904,B 24.9436,C -1.7345,E1 24.9909,E2 -176.979} C_DIS
LIN {X -8.535,Y -99.7846,Z 102,A -99.5914,B 24.9436,C -1.7344,E1 24.985,E2 -174.8767} C_DIS
LIN {X -12.1872,Y -99.4045,Z 102,A -101.8056,B 24.9439,C -1.7305,E1 24.9789,E2 -172.6519} C_DIS
LIN {X -15.9671,Y -98.8679,Z 102,A -104.2919,B 24.9446,C -1.7201,E1 24.9719,E2 -170.1386} C_DIS
LIN {X -19.5559,Y -98.2209,Z 102,A -105.704,B 24.9429,C -1.7454,E1 24.9682,E2 -168.7852} C_DIS
LIN {X -25.0555,Y -96.9625,Z 102,A -109.0397,B 24.9431,C -1.7432,E1 24.9591,E2 -165.4397} C_DIS
LIN {X -28.1154,Y -96.1206,Z 102,A -111.0018,B 24.9433,C -1.7391,E1 24.9538,E2 -163.4646} C_DIS
LIN {X -31.4933,Y -95.0681,Z 102,A -113.0611,B 24.9433,C -1.7393,E1 24.9483,E2 -161.4022} C_DIS
LIN {X -36.2872,Y -93.3427,Z 102,A -115.602,B 24.9422,C -1.7555,E1 24.9418,E2 -158.8945} C_DIS
LIN {X -40.552,Y -91.571,Z 102,A -118.4413,B 24.9425,C -1.7511,E1 24.9344,E2 -156.0383} C_DIS
LIN {X -44.4621,Y -89.7364,Z 102,A -120.8197,B 24.9421,C -1.7573,E1 24.9284,E2 -153.6687} C_DIS
LIN {X -46.8913,Y -88.4917,Z 102,A -122.59,B 24.9425,C -1.7519,E1 24.924,E2 -151.8806} C_DIS
LIN {X -51.4224,Y -85.9391,Z 102,A -125.3993,B 24.9418,C -1.762,E1 24.9172,E2 -149.0869} C_DIS
LIN {X -53.4681,Y -84.6811,Z 102,A -127.1927,B 24.9427,C -1.7493,E1 24.9129,E2 -147.2576} C_DIS
LIN {X -57.1161,Y -82.2633,Z 102,A -129.4252,B 24.9418,C -1.7629,E1 24.9078,E2 -145.05} C_DIS
LIN {X -59.8842,Y -80.2713,Z 102,A -131.3971,B 24.9416,C -1.7655,E1 24.9034,E2 -143.0774} C_DIS
LIN {X -62.5644,Y -78.2019,Z 102,A -133.4275,B 24.9416,C -1.7657,E1 24.8989,E2 -141.0401} C_DIS
LIN {X -66.2798,Y -75.0785,Z 102,A -136.1605,B 24.9411,C -1.7726,E1 24.8931,E2 -138.3129} C_DIS
LIN {X -68.6349,Y -72.9298,Z 102,A -137.9389,B 24.9408,C -1.7779,E1 24.8895,E2 -136.5398} C_DIS
LIN {X -71.2078,Y -70.4198,Z 102,A -139.9994,B 24.9405,C -1.7821,E1 24.8854,E2 -134.4806} C_DIS
LIN {X -74.8713,Y -66.511,Z 102,A -143.2454,B 24.9405,C -1.7827,E1 24.8792,E2 -131.2217} C_DIS
LIN {X -76.7551,Y -64.3298,Z 102,A -144.7729,B 24.9399,C -1.7906,E1 24.8765,E2 -129.7061} C_DIS
LIN {X -78.8606,Y -61.7311,Z 102,A -146.7495,B 24.9397,C -1.793,E1 24.8731,E2 -127.7259} C_DIS
LIN {X -80.9397,Y -58.9773,Z 102,A -148.6364,B 24.9392,C -1.8009,E1 24.8699,E2 -125.8486} C_DIS
LIN {X -82.8129,Y -56.3166,Z 102,A -150.972,B 24.94,C -1.7894,E1 24.8662,E2 -123.4742} C_DIS
LIN {X -84.6724,Y -53.4821,Z 102,A -152.8778,B 24.9396,C -1.7956,E1 24.8633,E2 -121.5735} C_DIS
LIN {X -86.8267,Y -49.9062,Z 102,A -154.8698,B 24.9382,C -1.8154,E1 24.8606,E2 -119.6184} C_DIS
LIN {X -88.6535,Y -46.5839,Z 102,A -156.861,B 24.9374,C -1.8274,E1 24.8579,E2 -117.6452} C_DIS
LIN {X -90.013,Y -43.9034,Z 102,A -158.8373,B 24.9377,C -1.8234,E1 24.8555,E2 -115.6487} C_DIS
LIN {X -92.2177,Y -39.0567,Z 102,A -161.5469,B 24.9363,C -1.8435,E1 24.8524,E2 -112.9722} C_DIS
LIN {X -93.8586,Y -34.9341,Z 102,A -164.2667,B 24.9363,C -1.8447,E1 24.8496,E2 -110.2401} C_DIS
LIN {X -95.2476,Y -30.9419,Z 102,A -166.8653,B 24.9361,C -1.8459,E1 24.8473,E2 -107.6295} C_DIS
LIN {X -96.314,Y -27.4434,Z 102,A -168.9284,B 24.9356,C -1.8532,E1 24.8456,E2 -105.5719} C_DIS
LIN {X -97.2022,Y -24.1119,Z 102,A -171.1232,B 24.9357,C -1.8518,E1 24.8441,E2 -103.361} C_DIS
LIN {X -97.9469,Y -20.8837,Z 102,A -172.785,B 24.9348,C -1.8655,E1 24.8431,E2 -101.722} C_DIS
LIN {X -98.5659,Y -17.7275,Z 102,A -174.6649,B 24.9345,C -1.8699,E1 24.8421,E2 -99.8416} C_DIS
LIN {X -99.1748,Y -13.9243,Z 102,A -176.7619,B 24.9337,C -1.8804,E1 24.8412,E2 -97.7571} C_DIS
LIN {X -99.7742,Y -8.6548,Z 102,A -179.7942,B 24.933,C -1.8901,E1 24.8403,E2 -94.7297} C_DIS
LIN {X -100.0315,Y -4.8481,Z 102,A 177.542,B 24.9337,C -1.8811,E1 24.8399,E2 -92.0283} C_DIS
LIN {X -100.1465,Y -0.4498,Z 102,A 174.8338,B 24.9335,C -1.8829,E1 24.8398,E2 -89.3082} C_DIS
LIN {X -100.1049,Y 2.9211,Z 102,A 173.3319,B 24.9321,C -1.9032,E1 24.8399,E2 -87.8457} C_DIS
LIN {X -99.8416,Y 7.8212,Z 102,A 170.4992,B 24.9315,C -1.9114,E1 24.8404,E2 -85.0156} C_DIS
LIN {X -99.4565,Y 11.7439,Z 102,A 168.286,B 24.9309,C -1.9201,E1 24.841,E2 -82.8098} C_DIS
LIN {X -99.0485,Y 14.8036,Z 102,A 166.4678,B 24.9306,C -1.924,E1 24.8417,E2 -80.9902} C_DIS
LIN {X -98.5349,Y 17.8999,Z 102,A 164.4623,B 24.9306,C -1.9228,E1 24.8427,E2 -78.9699} C_DIS
LIN {X -97.9663,Y 20.7945,Z 102,A 162.8284,B 24.9302,C -1.93,E1 24.8437,E2 -77.3434} C_DIS
LIN {X -97.0816,Y 24.5923,Z 102,A 160.6832,B 24.9294,C -1.9399,E1 24.8451,E2 -75.2093} C_DIS
LIN {X -96.1864,Y 27.8923,Z 102,A 158.6918,B 24.9291,C -1.9449,E1 24.8466,E2 -73.2183} C_DIS
LIN {X -94.733,Y 32.4842,Z 102,A 155.8406,B 24.9287,C -1.9503,E1 24.849,E2 -70.3638} C_DIS
LIN {X -93.4447,Y 36.0269,Z 102,A 153.5827,B 24.9284,C -1.9536,E1 24.8513,E2 -68.1009} C_DIS
LIN {X -91.9607,Y 39.6597,Z 102,A 151.517,B 24.9275,C -1.9664,E1 24.8535,E2 -66.0543} C_DIS
LIN {X -90.6022,Y 42.6726,Z 102,A 149.7691,B 24.9267,C -1.9769,E1 24.8555,E2 -64.3218} C_DIS
LIN {X -89.1199,Y 45.6854,Z 102,A 147.4464,B 24.9273,C -1.9692,E1 24.8584,E2 -61.9683} C_DIS
LIN {X -86.5203,Y 50.4391,Z 102,A 144.7008,B 24.9257,C -1.99,E1 24.8621,E2 -59.258} C_DIS
LIN {X -84.3332,Y 54.0132,Z 102,A 141.7648,B 24.9266,C -1.9789,E1 24.8666,E2 -56.2804} C_DIS
LIN {X -82.5304,Y 56.7319,Z 102,A 139.7092,B 24.9266,C -1.9777,E1 24.8698,E2 -54.2119} C_DIS
LIN {X -80.3213,Y 59.8168,Z 102,A 137.997,B 24.9251,C -1.9989,E1 24.8726,E2 -52.542} C_DIS
LIN {X -77.4916,Y 63.441,Z 102,A 135.5786,B 24.924,C -2.013,E1 24.8768,E2 -50.1458} C_DIS
LIN {X -75.4698,Y 65.8317,Z 102,A 133.654,B 24.924,C -2.0131,E1 24.8803,E2 -48.2128} C_DIS
LIN {X -72.2501,Y 69.3503,Z 102,A 131.0498,B 24.9232,C -2.0241,E1 24.8852,E2 -45.6234} C_DIS
LIN {X -69.4614,Y 72.143,Z 102,A 128.8489,B 24.9226,C -2.0315,E1 24.8895,E2 -43.4307} C_DIS
LIN {X -67.5488,Y 73.9372,Z 102,A 127.054,B 24.9231,C -2.025,E1 24.8933,E2 -41.6129} C_DIS
LIN {X -63.6274,Y 77.3388,Z 102,A 124.275,B 24.9221,C -2.0381,E1 24.8991,E2 -38.8545} C_DIS
LIN {X -61.4845,Y 79.0528,Z 102,A 122.1343,B 24.9233,C -2.022,E1 24.9039,E2 -36.6676} C_DIS
LIN {X -58.8357,Y 81.0433,Z 102,A 119.8359,B 24.9241,C -2.0123,E1 24.9092,E2 -34.3379} C_DIS
LIN {X -54.8878,Y 83.767,Z 102,A 118.1814,B 24.9208,C -2.0548,E1 24.9128,E2 -32.7793} C_DIS
LIN {X -52.8641,Y 85.0584,Z 102,A 116.3012,B 24.922,C -2.04,E1 24.9174,E2 -30.8577} C_DIS
LIN {X -49.3418,Y 87.1506,Z 102,A 114.2598,B 24.9208,C -2.0545,E1 24.9222,E2 -28.8449} C_DIS
LIN {X -46.8785,Y 88.4984,Z 102,A 112.5796,B 24.9208,C -2.0547,E1 24.9264,E2 -27.1606} C_DIS
LIN {X -43.8167,Y 90.0547,Z 102,A 110.6363,B 24.9205,C -2.0587,E1 24.9312,E2 -25.2214} C_DIS
LIN {X -41.2553,Y 91.2552,Z 102,A 108.3737,B 24.9221,C -2.0388,E1 24.9371,E2 -22.906} C_DIS
LIN {X -37.6425,Y 92.8039,Z 102,A 106.7598,B 24.9201,C -2.064,E1 24.9411,E2 -21.3484} C_DIS
LIN {X -34.2891,Y 94.0944,Z 102,A 104.3235,B 24.9209,C -2.0534,E1 24.9476,E2 -18.8818} C_DIS
LIN {X -30.2113,Y 95.4835,Z 102,A 102.03,B 24.9202,C -2.0623,E1 24.9536,E2 -16.6053} C_DIS
LIN {X -26.2835,Y 96.637,Z 102,A 99.3502,B 24.921,C -2.0529,E1 24.9609,E2 -13.899} C_DIS
LIN {X -22.8637,Y 97.5031,Z 102,A 97.9034,B 24.9193,C -2.075,E1 24.9647,E2 -12.5026} C_DIS
LIN {X -17.0712,Y 98.6833,Z 102,A 94.5672,B 24.9189,C -2.0793,E1 24.9738,E2 -9.1731} C_DIS
LIN {X -10.4489,Y 99.6008,Z 102,A 90.8173,B 24.9185,C -2.0844,E1 24.9842,E2 -5.4323} C_DIS
LIN {X -4.636,Y 100.0406,Z 102,A 87.205,B 24.9192,C -2.0758,E1 24.9943,E2 -1.7982} C_DIS
LIN {X 1.6795,Y 100.1334,Z 102,A 83.0436,B 24.9207,C -2.0568,E1 25.006,E2 2.4081} C_DIS
LIN {X 5.5999,Y 99.9907,Z 102,A 81.5561,B 24.9185,C -2.0843,E1 25.01,E2 3.8299} C_DIS
LIN {X 8.0962,Y 99.8197,Z 102,A 79.2245,B 24.9211,C -2.0515,E1 25.0167,E2 6.238} C_DIS
LIN {X 12.5631,Y 99.3567,Z 102,A 77.2496,B 24.9194,C -2.0726,E1 25.022,E2 8.1615} C_DIS
LIN {X 16.468,Y 98.7841,Z 102,A 75.2948,B 24.9186,C -2.083,E1 25.0273,E2 10.0895} C_DIS
LIN {X 19.1307,Y 98.3034,Z 102,A 73.1994,B 24.9202,C -2.0623,E1 25.0332,E2 12.2317} C_DIS
LIN {X 23.9766,Y 97.2352,Z 102,A 70.8636,B 24.9189,C -2.0793,E1 25.0395,E2 14.5239} C_DIS
LIN {X 26.6273,Y 96.5441,Z 102,A 69.1683,B 24.9194,C -2.0735,E1 25.0441,E2 16.2302} C_DIS
LIN {X 29.6403,Y 95.6606,Z 102,A 67.4823,B 24.9192,C -2.0763,E1 25.0485,E2 17.9066} C_DIS
LIN {X 33.8383,Y 94.2588,Z 102,A 65.04,B 24.9191,C -2.0775,E1 25.055,E2 20.3413} C_DIS
LIN {X 36.4638,Y 93.2733,Z 102,A 63.305,B 24.9196,C -2.0711,E1 25.0595,E2 22.0878} C_DIS
LIN {X 39.1413,Y 92.182,Z 102,A 61.1759,B 24.9211,C -2.0515,E1 25.0651,E2 24.2583} C_DIS
LIN {X 42.1852,Y 90.829,Z 102,A 59.783,B 24.9198,C -2.0685,E1 25.0686,E2 25.6073} C_DIS
LIN {X 44.9971,Y 89.4712,Z 102,A 57.3637,B 24.9218,C -2.0424,E1 25.0747,E2 28.0819} C_DIS
LIN {X 48.3824,Y 87.6864,Z 102,A 55.7039,B 24.9205,C -2.0594,E1 25.0787,E2 29.6967} C_DIS
LIN {X 51.1873,Y 86.078,Z 102,A 53.7876,B 24.9209,C -2.0542,E1 25.0833,E2 31.6195} C_DIS
LIN {X 54.0213,Y 84.3279,Z 102,A 51.8274,B 24.9213,C -2.0492,E1 25.088,E2 33.5853} C_DIS
LIN {X 56.6951,Y 82.556,Z 102,A 50.1806,B 24.9209,C -2.0533,E1 25.0917,E2 35.2168} C_DIS
LIN {X 59.5114,Y 80.5486,Z 102,A 48.2784,B 24.9209,C -2.0528,E1 25.096,E2 37.1133} C_DIS
LIN {X 63.4556,Y 77.48,Z 102,A 45.4076,B 24.9214,C -2.0471,E1 25.1023,E2 39.987} C_DIS
LIN {X 65.8767,Y 75.4305,Z 102,A 43.5704,B 24.9218,C -2.0427,E1 25.1062,E2 41.8274} C_DIS
LIN {X 67.8239,Y 73.6848,Z 102,A 41.9939,B 24.9222,C -2.0366,E1 25.1095,E2 43.412} C_DIS
LIN {X 70.5944,Y 71.0354,Z 102,A 39.7858,B 24.9226,C -2.0314,E1 25.1139,E2 45.6231} C_DIS
LIN {X 73.1275,Y 68.4246,Z 102,A 37.5505,B 24.9234,C -2.0209,E1 25.1182,E2 47.8737} C_DIS
LIN {X 75.7005,Y 65.5676,Z 102,A 35.5889,B 24.9231,C -2.0251,E1 25.1218,E2 49.8165} C_DIS
LIN {X 78.4118,Y 62.2989,Z 102,A 33.5054,B 24.9225,C -2.0329,E1 25.1255,E2 51.8718} C_DIS
LIN {X 79.8901,Y 60.3917,Z 102,A 31.782,B 24.9238,C -2.0161,E1 25.1284,E2 53.6268} C_DIS
LIN {X 82.1569,Y 57.2691,Z 102,A 29.4306,B 24.9246,C -2.0049,E1 25.1323,E2 55.9932} C_DIS
LIN {X 84.4593,Y 53.8167,Z 102,A 27.3679,B 24.9242,C -2.011,E1 25.1354,E2 58.0312} C_DIS
LIN {X 86.1692,Y 51.033,Z 102,A 24.7655,B 24.9267,C -1.9772,E1 25.1392,E2 60.6999} C_DIS
LIN {X 88.2293,Y 47.3842,Z 102,A 23.175,B 24.9248,C -2.0024,E1 25.1413,E2 62.2227} C_DIS
LIN {X 89.2893,Y 45.3539,Z 102,A 21.7437,B 24.9254,C -1.994,E1 25.1431,E2 63.6663} C_DIS
LIN {X 91.5081,Y 40.6942,Z 102,A 18.8293,B 24.926,C -1.9871,E1 25.1465,E2 66.5811} C_DIS
LIN {X 92.8777,Y 37.461,Z 102,A 16.7355,B 24.9266,C -1.9779,E1 25.1488,E2 68.6851} C_DIS
LIN {X 94.5038,Y 33.1442,Z 102,A 14.2803,B 24.9266,C -1.9775,E1 25.1511,E2 71.1277} C_DIS
LIN {X 95.4697,Y 30.2555,Z 102,A 12.5149,B 24.9271,C -1.9713,E1 25.1527,E2 72.8976} C_DIS
LIN {X 96.5592,Y 26.5714,Z 102,A 9.5644,B 24.9298,C -1.9347,E1 25.155,E2 75.9175} C_DIS
LIN {X 97.6066,Y 22.4159,Z 102,A 8.2639,B 24.927,C -1.9731,E1 25.1558,E2 77.12} C_DIS
LIN {X 98.0884,Y 20.2034,Z 102,A 6.3686,B 24.9291,C -1.945,E1 25.1569,E2 79.0706} C_DIS
LIN {X 99.059,Y 14.7356,Z 102,A 3.4177,B 24.9291,C -1.944,E1 25.1582,E2 82.0064} C_DIS
LIN {X 99.5513,Y 10.9221,Z 102,A 1.3744,B 24.9291,C -1.9433,E1 25.1589,E2 84.0393} C_DIS
LIN {X 99.8894,Y 7.1977,Z 102,A -0.9495,B 24.9302,C -1.9291,E1 25.1595,E2 86.383} C_DIS
LIN {X 100.0693,Y 3.9676,Z 102,A -2.7008,B 24.9304,C -1.9271,E1 25.1597,E2 88.1285} C_DIS
LIN {X 100.1464,Y 0.468,Z 102,A -4.7406,B 24.9309,C -1.9192,E1 25.1597,E2 90.175} C_DIS
LIN {X 100.098,Y -3.1441,Z 102,A -6.8384,B 24.9315,C -1.9113,E1 25.1597,E2 92.2789} C_DIS
LIN {X 99.9204,Y -6.7382,Z 102,A -8.5848,B 24.9311,C -1.9172,E1 25.1594,E2 94.0009} C_DIS
LIN {X 99.3779,Y -12.3998,Z 102,A -11.8931,B 24.932,C -1.9044,E1 25.1585,E2 97.3198} C_DIS
LIN {X 98.4418,Y -18.412,Z 102,A -15.381,B 24.9328,C -1.8929,E1 25.1569,E2 100.8144} C_DIS
LIN {X 97.3743,Y -23.4064,Z 102,A -18.1829,B 24.9332,C -1.8884,E1 25.1553,E2 103.6106} C_DIS
LIN {X 96.5021,Y -26.7793,Z 102,A -21.2223,B 24.9365,C -1.8401,E1 25.153,E2 106.7463} C_DIS
LIN {X 95.1306,Y -31.3035,Z 102,A -22.9448,B 24.9344,C -1.8709,E1 25.1516,E2 108.3866} C_DIS
LIN {X 93.9148,Y -34.7815,Z 102,A -25.6532,B 24.9365,C -1.8403,E1 25.1489,E2 111.152} C_DIS
LIN {X 92.7039,Y -37.888,Z 102,A -27.5598,B 24.9369,C -1.8345,E1 25.1469,E2 113.0618} C_DIS
LIN {X 91.3465,Y -41.0528,Z 102,A -28.7289,B 24.9351,C -1.8606,E1 25.1457,E2 114.1629} C_DIS
LIN {X 90.2707,Y -43.367,Z 102,A -30.4898,B 24.9363,C -1.844,E1 25.1436,E2 115.9533} C_DIS
LIN {X 86.9409,Y -49.7074,Z 102,A -34.2553,B 24.9362,C -1.8452,E1 25.1387,E2 119.6962} C_DIS
LIN {X 85.325,Y -52.4346,Z 102,A -36.2885,B 24.9371,C -1.8312,E1 25.1357,E2 121.7522} C_DIS
LIN {X 82.1689,Y -57.2518,Z 102,A -39.28,B 24.937,C -1.834,E1 25.1312,E2 124.722} C_DIS
LIN {X 79.7041,Y -60.6386,Z 102,A -41.8822,B 24.938,C -1.8192,E1 25.1268,E2 127.3467} C_DIS
LIN {X 75.6263,Y -65.6524,Z 102,A -45.6577,B 24.9388,C -1.8063,E1 25.1201,E2 131.1351} C_DIS
LIN {X 73.5591,Y -67.9608,Z 102,A -47.3702,B 24.939,C -1.8042,E1 25.1169,E2 132.8451} C_DIS
LIN {X 72.1046,Y -69.5012,Z 102,A -48.6633,B 24.9394,C -1.798,E1 25.1144,E2 134.1473} C_DIS
LIN {X 67.9892,Y -73.5328,Z 102,A -51.9971,B 24.94,C -1.7886,E1 25.1077,E2 137.4895} C_DIS
LIN {X 65.5259,Y -75.7363,Z 102,A -53.7027,B 24.9398,C -1.7915,E1 25.1041,E2 139.1813} C_DIS
LIN {X 63.8119,Y -77.1855,Z 102,A -55.2009,B 24.9406,C -1.7802,E1 25.1008,E2 140.7005} C_DIS
LIN {X 57.7684,Y -81.808,Z 102,A -60.1666,B 24.9428,C -1.7472,E1 25.0896,E2 145.7264} C_DIS
LIN {X 54.1688,Y -84.2333,Z 102,A -61.5336,B 24.9402,C -1.7858,E1 25.0866,E2 146.9977} C_DIS
LIN {X 50.3089,Y -86.5953,Z 102,A -64.9189,B 24.9426,C -1.7499,E1 25.0783,E2 150.4573} C_DIS
LIN {X 47.5123,Y -88.1598,Z 102,A -66.9056,B 24.9432,C -1.7409,E1 25.0734,E2 152.4597} C_DIS
LIN {X 44.0391,Y -89.9461,Z 102,A -68.5586,B 24.942,C -1.7596,E1 25.0694,E2 154.064} C_DIS
LIN {X 37.7241,Y -92.7706,Z 102,A -72.047,B 24.9412,C -1.7718,E1 25.0606,E2 157.515} C_DIS
LIN {X 35.5033,Y -93.643,Z 102,A -73.8398,B 24.9424,C -1.7533,E1 25.0558,E2 159.3475} C_DIS
LIN {X 30.7571,Y -95.3074,Z 102,A -76.6993,B 24.9426,C -1.7504,E1 25.0482,E2 162.2084} C_DIS
LIN {X 26.5636,Y -96.5613,Z 102,A -79.0361,B 24.9423,C -1.7539,E1 25.042,E2 164.5328} C_DIS
LIN {X 24.2275,Y -97.174,Z 102,A -81.3911,B 24.9448,C -1.7157,E1 25.0354,E2 166.9748} C_DIS
LIN {X 19.7122,Y -98.1892,Z 102,A -83.1918,B 24.9429,C -1.7453,E1 25.0307,E2 168.7032} C_DIS
LIN {X 12.2494,Y -99.3973,Z 102,A -87.4514,B 24.9429,C -1.7446,E1 25.0189,E2 172.9604} C_DIS
LIN {X 9.3812,Y -99.7072,Z 102,A -89.5279,B 24.9441,C -1.7277,E1 25.013,E2 175.0756} C_DIS
LIN {X 3.6862,Y -100.0814,Z 102,A -92.5478,B 24.9436,C -1.7355,E1 25.0047,E2 178.0759} C_DIS
LIN {X 0.6945,Y -100.1423,Z 102,A -93.5311,B 24.9418,C -1.7624,E1 25.0021,E2 178.9953} C_DIS
Enddeposition()
LIN {X 0.6945,Y -100.1423,Z 102,A -93.5311,B 24.9418,C -1.7624,E1 25.0021,E2 178.9953} C_DIS
Startdeposition()
$VEL.CP = VEL_PRINT
LIN {X 1.8164,Y -99.2685,Z 102,A -92.7045,B 24.9403,C -1.7842,E1 25.0046,E2 178.117} C_DIS
LIN {X 6.7084,Y -99.0583,Z 102,A -89.4529,B 24.9392,C -1.8015,E1 25.0137,E2 174.8258} C_DIS
LIN {X 9.9875,Y -98.7822,Z 102,A -87.9728,B 24.9402,C -1.7866,E1 25.0178,E2 173.3819} C_DIS
LIN {X 13.6514,Y -98.3427,Z 102,A -85.0685,B 24.9381,C -1.8176,E1 25.026,E2 170.4064} C_DIS
LIN {X 18.2488,Y -97.5951,Z 102,A -83.0646,B 24.9397,C -1.7935,E1 25.0313,E2 168.462} C_DIS
LIN {X 23.6823,Y -96.4195,Z 102,A -80.0506,B 24.94,C -1.789,E1 25.0395,E2 165.4626} C_DIS
LIN {X 26.7183,Y -95.6232,Z 102,A -78.1242,B 24.9396,C -1.7954,E1 25.0447,E2 163.5243} C_DIS
LIN {X 29.6586,Y -94.7522,Z 102,A -75.7097,B 24.9377,C -1.8225,E1 25.0513,E2 161.05} C_DIS
LIN {X 33.6939,Y -93.3937,Z 102,A -74.1099,B 24.9398,C -1.7923,E1 25.0553,E2 159.5248} C_DIS
LIN {X 36.3466,Y -92.393,Z 102,A -72.2855,B 24.9391,C -1.8019,E1 25.0601,E2 157.6817} C_DIS
LIN {X 40.7652,Y -90.5303,Z 102,A -69.5645,B 24.939,C -1.8042,E1 25.0671,E2 154.9618} C_DIS
LIN {X 43.851,Y -89.077,Z 102,A -67.5507,B 24.9387,C -1.8091,E1 25.0722,E2 152.9416} C_DIS
LIN {X 46.9686,Y -87.4739,Z 102,A -64.9216,B 24.9368,C -1.8364,E1 25.0788,E2 150.2554} C_DIS
LIN {X 50.5344,Y -85.4623,Z 102,A -63.2267,B 24.9383,C -1.8144,E1 25.0828,E2 148.6177} C_DIS
LIN {X 53.2375,Y -83.8065,Z 102,A -61.5917,B 24.9386,C -1.8103,E1 25.0866,E2 146.9977} C_DIS
LIN {X 55.6886,Y -82.1968,Z 102,A -59.7146,B 24.9379,C -1.8209,E1 25.091,E2 145.1018} C_DIS
LIN {X 58.6978,Y -80.0757,Z 102,A -57.8394,B 24.9382,C -1.8155,E1 25.0952,E2 143.246} C_DIS
LIN {X 61.6965,Y -77.7889,Z 102,A -55.3836,B 24.9371,C -1.8312,E1 25.1007,E2 140.7621} C_DIS
LIN {X 64.3904,Y -75.5739,Z 102,A -53.4211,B 24.937,C -1.8337,E1 25.1049,E2 138.8012} C_DIS
LIN {X 66.4285,Y -73.7894,Z 102,A -50.9261,B 24.9341,C -1.8746,E1 25.1103,E2 136.2196} C_DIS
LIN {X 70.2704,Y -70.1418,Z 102,A -48.7469,B 24.9361,C -1.8468,E1 25.1144,E2 134.1153} C_DIS
LIN {X 72.6216,Y -67.704,Z 102,A -46.7457,B 24.9356,C -1.8535,E1 25.1183,E2 132.1069} C_DIS
LIN {X 77.5347,Y -62.0181,Z 102,A -42.5432,B 24.9352,C -1.8594,E1 25.1258,E2 127.9096} C_DIS
LIN {X 79.3778,Y -59.6381,Z 102,A -40.8688,B 24.935,C -1.8616,E1 25.1287,E2 126.238} C_DIS
LIN {X 81.206,Y -57.1266,Z 102,A -39.1198,B 24.9348,C -1.8648,E1 25.1315,E2 124.49} C_DIS
LIN {X 82.6411,Y -55.029,Z 102,A -37.4225,B 24.9339,C -1.8782,E1 25.1342,E2 122.7696} C_DIS
LIN {X 84.6182,Y -51.9373,Z 102,A -35.4638,B 24.9339,C -1.8778,E1 25.1371,E2 120.8216} C_DIS
LIN {X 85.9898,Y -49.632,Z 102,A -33.6068,B 24.9327,C -1.8948,E1 25.1397,E2 118.9341} C_DIS
LIN {X 88.403,Y -45.1934,Z 102,A -31.1482,B 24.9334,C -1.8849,E1 25.1429,E2 116.5117} C_DIS
LIN {X 89.7617,Y -42.4349,Z 102,A -29.2899,B 24.9328,C -1.8936,E1 25.1451,E2 114.6429} C_DIS
LIN {X 91.0154,Y -39.6705,Z 102,A -27.5804,B 24.9325,C -1.8973,E1 25.1471,E2 112.9341} C_DIS
LIN {X 93.105,Y -34.4853,Z 102,A -24.4651,B 24.9321,C -1.9027,E1 25.1503,E2 109.8233} C_DIS
LIN {X 93.9344,Y -32.1571,Z 102,A -22.895,B 24.9314,C -1.913,E1 25.1517,E2 108.2378} C_DIS
LIN {X 95.2516,Y -28.013,Z 102,A -20.3619,B 24.9308,C -1.9218,E1 25.1538,E2 105.6982} C_DIS
LIN {X 96.0904,Y -24.9852,Z 102,A -18.6415,B 24.9306,C -1.9238,E1 25.155,E2 103.9829} C_DIS
LIN {X 96.8364,Y -21.919,Z 102,A -16.5734,B 24.9295,C -1.9397,E1 25.1563,E2 101.8895} C_DIS
LIN {X 97.688,Y -17.7374,Z 102,A -14.7172,B 24.9307,C -1.923,E1 25.1573,E2 100.0834} C_DIS
LIN {X 98.3356,Y -13.7013,Z 102,A -11.9874,B 24.929,C -1.9456,E1 25.1585,E2 97.3164} C_DIS
LIN {X 98.7667,Y -10.1349,Z 102,A -9.9341,B 24.9286,C -1.9515,E1 25.1591,E2 95.2614} C_DIS
LIN {X 99,Y -7.5297,Z 102,A -8.396,B 24.9282,C -1.9575,E1 25.1595,E2 93.7183} C_DIS
LIN {X 99.2197,Y -3.6553,Z 102,A -6.1757,B 24.9277,C -1.9639,E1 25.1597,E2 91.4959} C_DIS
LIN {X 99.2812,Y -0.9542,Z 102,A -4.3938,B 24.9266,C -1.978,E1 25.1597,E2 89.6914} C_DIS
LIN {X 99.2137,Y 3.796,Z 102,A -2.1142,B 24.9274,C -1.9681,E1 25.1597,E2 87.4487} C_DIS
LIN {X 99.0557,Y 6.7462,Z 102,A -0.3041,B 24.9267,C -1.9779,E1 25.1593,E2 85.6264} C_DIS
LIN {X 98.7507,Y 10.2879,Z 102,A 2.3891,B 24.9242,C -2.0105,E1 25.1585,E2 82.8722} C_DIS
LIN {X 98.2235,Y 14.49,Z 102,A 4.9812,B 24.9232,C -2.0242,E1 25.1575,E2 80.263} C_DIS
LIN {X 97.4127,Y 19.196,Z 102,A 6.9808,B 24.9248,C -2.0021,E1 25.1565,E2 78.3272} C_DIS
LIN {X 96.6574,Y 22.6938,Z 102,A 8.9079,B 24.9248,C -2.0029,E1 25.1553,E2 76.4093} C_DIS
LIN {X 96.1412,Y 24.7876,Z 102,A 10.3437,B 24.9239,C -2.0145,E1 25.1543,E2 74.9546} C_DIS
LIN {X 95.1637,Y 28.3094,Z 102,A 12.2481,B 24.924,C -2.0127,E1 25.1528,E2 73.0653} C_DIS
LIN {X 94.0438,Y 31.8325,Z 102,A 14.445,B 24.9234,C -2.0216,E1 25.1509,E2 70.8598} C_DIS
LIN {X 92.6685,Y 35.6419,Z 102,A 16.7992,B 24.9228,C -2.0291,E1 25.1486,E2 68.5009} C_DIS
LIN {X 91.6024,Y 38.2965,Z 102,A 18.1581,B 24.9233,C -2.0223,E1 25.1472,E2 67.1657} C_DIS
LIN {X 90.6982,Y 40.3927,Z 102,A 19.8401,B 24.9219,C -2.0406,E1 25.1452,E2 65.4497} C_DIS
LIN {X 88.9264,Y 44.1547,Z 102,A 21.9935,B 24.9222,C -2.0375,E1 25.1426,E2 63.315} C_DIS
LIN {X 87.464,Y 46.9867,Z 102,A 23.898,B 24.9216,C -2.0452,E1 25.1402,E2 61.4025} C_DIS
LIN {X 85.5446,Y 50.3953,Z 102,A 26.1073,B 24.9212,C -2.0494,E1 25.1371,E2 59.1948} C_DIS
LIN {X 83.8065,Y 53.2375,Z 102,A 28.0896,B 24.9207,C -2.0568,E1 25.1341,E2 57.2051} C_DIS
LIN {X 82.0306,Y 55.9337,Z 102,A 29.9813,B 24.9202,C -2.0627,E1 25.1312,E2 55.3087} C_DIS
LIN {X 80.1859,Y 58.5473,Z 102,A 31.7088,B 24.9202,C -2.0627,E1 25.1284,E2 53.5898} C_DIS
LIN {X 78.063,Y 61.3497,Z 102,A 33.6876,B 24.92,C -2.0656,E1 25.125,E2 51.6134} C_DIS
LIN {X 75.8807,Y 64.0304,Z 102,A 35.7774,B 24.9193,C -2.074,E1 25.1213,E2 49.5133} C_DIS
LIN {X 73.225,Y 67.0497,Z 102,A 38.0081,B 24.9193,C -2.0757,E1 25.1171,E2 47.2884} C_DIS
LIN {X 70.8283,Y 69.5771,Z 102,A 40.0389,B 24.9188,C -2.0809,E1 25.1132,E2 45.2542} C_DIS
LIN {X 68.3229,Y 72.0396,Z 102,A 42.0682,B 24.9185,C -2.0852,E1 25.1091,E2 43.2231} C_DIS
LIN {X 65.762,Y 74.3859,Z 102,A 44.1414,B 24.9179,C -2.0919,E1 25.1048,E2 41.1424} C_DIS
LIN {X 63.0165,Y 76.7254,Z 102,A 46.3359,B 24.9173,C -2.1003,E1 25.1,E2 38.9365} C_DIS
LIN {X 59.6032,Y 79.404,Z 102,A 48.6476,B 24.9175,C -2.0974,E1 25.095,E2 36.6402} C_DIS
LIN {X 57.1588,Y 81.1835,Z 102,A 50.4691,B 24.917,C -2.1033,E1 25.0908,E2 34.8111} C_DIS
LIN {X 54.6355,Y 82.9005,Z 102,A 52.0916,B 24.9172,C -2.1008,E1 25.0871,E2 33.1998} C_DIS
LIN {X 51.1166,Y 85.117,Z 102,A 54.3908,B 24.9172,C -2.1006,E1 25.0816,E2 30.9084} C_DIS
LIN {X 48.9703,Y 86.37,Z 102,A 56.048,B 24.9164,C -2.1111,E1 25.0776,E2 29.2312} C_DIS
LIN {X 45.6991,Y 88.1446,Z 102,A 58.0863,B 24.9165,C -2.1098,E1 25.0725,E2 27.2018} C_DIS
LIN {X 42.8183,Y 89.5778,Z 102,A 59.9566,B 24.9163,C -2.1127,E1 25.0678,E2 25.3297} C_DIS
LIN {X 40.414,Y 90.6886,Z 102,A 61.5767,B 24.9159,C -2.1179,E1 25.0637,E2 23.7012} C_DIS
LIN {X 36.8881,Y 92.18,Z 102,A 63.7891,B 24.9157,C -2.1203,E1 25.058,E2 21.4882} C_DIS
LIN {X 33.1586,Y 93.5849,Z 102,A 66.0101,B 24.9157,C -2.1194,E1 25.0522,E2 19.274} C_DIS
LIN {X 29.6808,Y 94.7453,Z 102,A 68.0984,B 24.9157,C -2.1201,E1 25.0466,E2 17.188} C_DIS
LIN {X 26.1033,Y 95.7925,Z 102,A 70.2589,B 24.9156,C -2.1219,E1 25.0408,E2 15.0267} C_DIS
LIN {X 22.9643,Y 96.5946,Z 102,A 72.1375,B 24.9154,C -2.1233,E1 25.0357,E2 13.1476} C_DIS
LIN {X 19.2274,Y 97.4067,Z 102,A 74.3545,B 24.9154,C -2.1247,E1 25.0297,E2 10.93} C_DIS
LIN {X 15.8435,Y 98.0144,Z 102,A 76.2196,B 24.9156,C -2.121,E1 25.0246,E2 9.0757} C_DIS
LIN {X 11.9686,Y 98.562,Z 102,A 78.4314,B 24.9157,C -2.1198,E1 25.0184,E2 6.8685} C_DIS
LIN {X 6.9578,Y 99.0414,Z 102,A 81.2166,B 24.9161,C -2.1157,E1 25.0107,E2 4.0947} C_DIS
LIN {X 3.1676,Y 99.2347,Z 102,A 83.6462,B 24.9154,C -2.1243,E1 25.0039,E2 1.6454} C_DIS
LIN {X -1.1863,Y 99.2776,Z 102,A 86.5367,B 24.9143,C -2.1376,E1 24.9957,E2 -1.2767} C_DIS
LIN {X -4.3885,Y 99.1882,Z 102,A 87.6266,B 24.9166,C -2.1094,E1 24.9929,E2 -2.2998} C_DIS
LIN {X -9.2369,Y 98.8546,Z 102,A 90.8998,B 24.9153,C -2.1251,E1 24.9837,E2 -5.6116} C_DIS
LIN {X -13.9422,Y 98.3014,Z 102,A 93.4965,B 24.9158,C -2.1185,E1 24.9765,E2 -8.1944} C_DIS
LIN {X -17.1222,Y 97.7987,Z 102,A 95.5187,B 24.9155,C -2.123,E1 24.9709,E2 -10.2294} C_DIS
LIN {X -21.8069,Y 96.8623,Z 102,A 98.2961,B 24.9155,C -2.1214,E1 24.9633,E2 -13.0061} C_DIS
LIN {X -25.7949,Y 95.8758,Z 102,A 100.5226,B 24.9162,C -2.1139,E1 24.9573,E2 -15.2182} C_DIS
LIN {X -29.2658,Y 94.874,Z 102,A 102.381,B 24.917,C -2.1036,E1 24.9524,E2 -17.0551} C_DIS
LIN {X -31.2031,Y 94.2561,Z 102,A 103.8805,B 24.9162,C -2.1137,E1 24.9484,E2 -18.5814} C_DIS
LIN {X -34.3942,Y 93.1383,Z 102,A 105.807,B 24.9165,C -2.1104,E1 24.9433,E2 -20.5038} C_DIS
LIN {X -37.652,Y 91.8691,Z 102,A 107.8879,B 24.9165,C -2.1098,E1 24.9379,E2 -22.588} C_DIS
LIN {X -41.1678,Y 90.3489,Z 102,A 110.0813,B 24.9168,C -2.1059,E1 24.9323,E2 -24.7773} C_DIS
LIN {X -44.6163,Y 88.6976,Z 102,A 112.361,B 24.9169,C -2.1049,E1 24.9266,E2 -27.0608} C_DIS
LIN {X -48.148,Y 86.8297,Z 102,A 114.5398,B 24.9176,C -2.0966,E1 24.9213,E2 -29.2259} C_DIS
LIN {X -51.2329,Y 85.0463,Z 102,A 116.7756,B 24.9174,C -2.0991,E1 24.9159,E2 -31.4745} C_DIS
LIN {X -54.6365,Y 82.8999,Z 102,A 118.9117,B 24.9182,C -2.0882,E1 24.9109,E2 -33.5915} C_DIS
LIN {X -58.2017,Y 80.4389,Z 102,A 122.1829,B 24.9165,C -2.11,E1 24.9034,E2 -36.9259} C_DIS
LIN {X -61.7227,Y 77.7682,Z 102,A 123.984,B 24.919,C -2.0785,E1 24.8996,E2 -38.6587} C_DIS
LIN {X -64.8414,Y 75.1897,Z 102,A 126.44,B 24.919,C -2.0774,E1 24.8943,E2 -41.1216} C_DIS
LIN {X -67.543,Y 72.7723,Z 102,A 128.4976,B 24.9195,C -2.0714,E1 24.8901,E2 -43.1732} C_DIS
LIN {X -69.7734,Y 70.6344,Z 102,A 130.2939,B 24.9198,C -2.0676,E1 24.8865,E2 -44.968} C_DIS
LIN {X -72.6364,Y 67.6882,Z 102,A 132.701,B 24.9202,C -2.063,E1 24.8818,E2 -47.3745} C_DIS
LIN {X -75.1005,Y 64.9437,Z 102,A 134.834,B 24.9206,C -2.0577,E1 24.8779,E2 -49.5045} C_DIS
LIN {X -77.0793,Y 62.5806,Z 102,A 136.4008,B 24.9215,C -2.0459,E1 24.8752,E2 -51.0504} C_DIS
LIN {X -79.0758,Y 60.0402,Z 102,A 138.9779,B 24.92,C -2.0652,E1 24.8707,E2 -53.6856} C_DIS
LIN {X -81.2685,Y 57.0366,Z 102,A 140.3782,B 24.9224,C -2.034,E1 24.8685,E2 -55.0184} C_DIS
LIN {X -83.0874,Y 54.3521,Z 102,A 142.4163,B 24.9224,C -2.0344,E1 24.8654,E2 -57.0675} C_DIS
LIN {X -84.7144,Y 51.779,Z 102,A 144.3087,B 24.9224,C -2.034,E1 24.8626,E2 -58.9687} C_DIS
LIN {X -86.553,Y 48.6436,Z 102,A 146.3548,B 24.923,C -2.0262,E1 24.8597,E2 -61.0068} C_DIS
LIN {X -88.7355,Y 44.5399,Z 102,A 148.9669,B 24.9238,C -2.0159,E1 24.8564,E2 -63.6083} C_DIS
LIN {X -89.8361,Y 42.2751,Z 102,A 150.5754,B 24.9238,C -2.0167,E1 24.8544,E2 -65.2276} C_DIS
LIN {X -91.4159,Y 38.739,Z 102,A 152.8079,B 24.9243,C -2.0099,E1 24.8519,E2 -67.4561} C_DIS
LIN {X -93.1323,Y 34.4105,Z 102,A 155.2403,B 24.9255,C -1.9931,E1 24.8495,E2 -69.8621} C_DIS
LIN {X -94.944,Y 29.0401,Z 102,A 158.8298,B 24.9255,C -1.9935,E1 24.8464,E2 -73.473} C_DIS
LIN {X -95.7529,Y 26.2499,Z 102,A 160.3292,B 24.9263,C -1.9823,E1 24.8452,E2 -74.9544} C_DIS
LIN {X -96.5242,Y 23.2532,Z 102,A 162.1251,B 24.9267,C -1.977,E1 24.844,E2 -76.7481} C_DIS
LIN {X -97.1847,Y 20.3177,Z 102,A 164.076,B 24.9266,C -1.9786,E1 24.8429,E2 -78.7144} C_DIS
LIN {X -97.8133,Y 17.0412,Z 102,A 166.0502,B 24.9269,C -1.974,E1 24.8419,E2 -80.6894} C_DIS
LIN {X -98.3876,Y 13.3323,Z 102,A 167.9772,B 24.928,C -1.9591,E1 24.8411,E2 -82.5923} C_DIS
LIN {X -98.7399,Y 10.3911,Z 102,A 169.6975,B 24.9284,C -1.954,E1 24.8406,E2 -84.3106} C_DIS
LIN {X -98.9998,Y 7.5322,Z 102,A 171.4012,B 24.9287,C -1.9502,E1 24.8402,E2 -86.0155} C_DIS
LIN {X -99.1946,Y 4.24,Z 102,A 173.3705,B 24.929,C -1.9463,E1 24.8399,E2 -87.9873} C_DIS
LIN {X -99.2811,Y 0.9578,Z 102,A 175.5537,B 24.9287,C -1.9498,E1 24.8398,E2 -90.1922} C_DIS
LIN {X -99.2238,Y -3.5239,Z 102,A 177.8271,B 24.9301,C -1.931,E1 24.8399,E2 -92.4343} C_DIS
LIN {X -99.0537,Y -6.7754,Z 102,A 179.8987,B 24.9301,C -1.9315,E1 24.8403,E2 -94.5195} C_DIS
LIN {X -98.7372,Y -10.4166,Z 102,A -177.8786,B 24.9303,C -1.9286,E1 24.8409,E2 -96.7486} C_DIS
LIN {X -98.2674,Y -14.1809,Z 102,A -175.7743,B 24.931,C -1.9188,E1 24.8417,E2 -98.8422} C_DIS
LIN {X -97.6258,Y -18.0834,Z 102,A -173.6281,B 24.9318,C -1.907,E1 24.8427,E2 -100.973} C_DIS
LIN {X -96.9907,Y -21.2213,Z 102,A -171.8157,B 24.9323,C -1.9001,E1 24.8437,E2 -102.7796} C_DIS
LIN {X -96.2603,Y -24.3239,Z 102,A -169.7924,B 24.9323,C -1.9007,E1 24.8451,E2 -104.8161} C_DIS
LIN {X -95.3023,Y -27.8422,Z 102,A -167.7888,B 24.933,C -1.8909,E1 24.8466,E2 -106.8079} C_DIS
LIN {X -94.3964,Y -30.7719,Z 102,A -165.8638,B 24.933,C -1.8909,E1 24.8482,E2 -108.7438} C_DIS
LIN {X -93.2254,Y -34.1554,Z 102,A -163.8892,B 24.9336,C -1.8816,E1 24.8501,E2 -110.7077} C_DIS
LIN {X -92.1441,Y -36.9762,Z 102,A -162.0788,B 24.9338,C -1.8788,E1 24.8519,E2 -112.5214} C_DIS
LIN {X -90.8704,Y -40.0031,Z 102,A -160.0999,B 24.934,C -1.8762,E1 24.8541,E2 -114.5052} C_DIS
LIN {X -89.2649,Y -43.4695,Z 102,A -158.097,B 24.9349,C -1.8631,E1 24.8565,E2 -116.4877} C_DIS
LIN {X -87.7485,Y -46.452,Z 102,A -155.9515,B 24.9348,C -1.8651,E1 24.8593,E2 -118.6495} C_DIS
LIN {X -86.0952,Y -49.4486,Z 102,A -154.2451,B 24.9358,C -1.8506,E1 24.8616,E2 -120.3303} C_DIS
LIN {X -84.6293,Y -51.9191,Z 102,A -152.3692,B 24.9356,C -1.8537,E1 24.8643,E2 -122.2231} C_DIS
LIN {X -83.1152,Y -54.31,Z 102,A -150.5848,B 24.9356,C -1.8546,E1 24.867,E2 -124.0188} C_DIS
LIN {X -81.2022,Y -57.132,Z 102,A -148.66,B 24.936,C -1.8482,E1 24.8701,E2 -125.9378} C_DIS
LIN {X -79.0806,Y -60.0338,Z 102,A -146.6954,B 24.9366,C -1.8393,E1 24.8733,E2 -127.8907} C_DIS
LIN {X -77.0725,Y -62.589,Z 102,A -144.9941,B 24.9373,C -1.8289,E1 24.8763,E2 -129.5751} C_DIS
LIN {X -71.8267,Y -68.5471,Z 102,A -140.0988,B 24.9373,C -1.8294,E1 24.8854,E2 -134.4934} C_DIS
LIN {X -69.2898,Y -71.1108,Z 102,A -138.0773,B 24.9377,C -1.8229,E1 24.8894,E2 -136.5079} C_DIS
LIN {X -66.7832,Y -73.4695,Z 102,A -136.1601,B 24.9382,C -1.8165,E1 24.8933,E2 -138.4176} C_DIS
LIN {X -64.3644,Y -75.596,Z 102,A -134.1761,B 24.9381,C -1.8173,E1 24.8975,E2 -140.4114} C_DIS
LIN {X -61.6943,Y -77.7906,Z 102,A -132.2496,B 24.9385,C -1.8112,E1 24.9017,E2 -142.3306} C_DIS
LIN {X -59.1691,Y -79.7302,Z 102,A -130.2535,B 24.9384,C -1.8135,E1 24.9062,E2 -144.3395} C_DIS
LIN {X -56.2418,Y -81.821,Z 102,A -127.7233,B 24.9375,C -1.8263,E1 24.9121,E2 -146.9086} C_DIS
LIN {X -53.0441,Y -83.9293,Z 102,A -126.1805,B 24.9393,C -1.7991,E1 24.9156,E2 -148.3916} C_DIS
LIN {X -50.4944,Y -85.486,Z 102,A -124.3845,B 24.9393,C -1.7991,E1 24.9199,E2 -150.1932} C_DIS
LIN {X -47.4815,Y -87.1956,Z 102,A -122.5247,B 24.9399,C -1.7914,E1 24.9244,E2 -152.0401} C_DIS
LIN {X -45.1014,Y -88.4501,Z 102,A -120.74,B 24.9394,C -1.7977,E1 24.9289,E2 -153.8446} C_DIS
LIN {X -41.4099,Y -90.2389,Z 102,A -118.5841,B 24.9401,C -1.7873,E1 24.9343,E2 -155.9812} C_DIS
LIN {X -37.955,Y -91.7457,Z 102,A -116.1153,B 24.9396,C -1.7956,E1 24.9407,E2 -158.4755} C_DIS
LIN {X -35.296,Y -92.7995,Z 102,A -114.5903,B 24.94,C -1.7895,E1 24.9446,E2 -159.9893} C_DIS
LIN {X -31.9361,Y -94.0089,Z 102,A -112.7461,B 24.9406,C -1.7799,E1 24.9494,E2 -161.8142} C_DIS
LIN {X -29.3257,Y -94.8554,Z 102,A -110.884,B 24.94,C -1.7888,E1 24.9544,E2 -163.7009} C_DIS
LIN {X -26.3871,Y -95.7159,Z 102,A -109.1113,B 24.94,C -1.7879,E1 24.9592,E2 -165.4741} C_DIS
LIN {X -23.9104,Y -96.3638,Z 102,A -107.5202,B 24.9399,C -1.7912,E1 24.9635,E2 -167.0754} C_DIS
LIN {X -20.1552,Y -97.218,Z 102,A -105.4977,B 24.9404,C -1.7829,E1 24.969,E2 -169.0805} C_DIS
LIN {X -17.8589,Y -97.6662,Z 102,A -103.9582,B 24.94,C -1.7894,E1 24.9733,E2 -170.6371} C_DIS
LIN {X -11.4108,Y -98.6274,Z 102,A -100.2939,B 24.9403,C -1.7849,E1 24.9834,E2 -174.2936} C_DIS
LIN {X -7.8354,Y -98.9755,Z 102,A -98.246,B 24.9403,C -1.7838,E1 24.9891,E2 -176.3401} C_DIS
LIN {X -4.7427,Y -99.173,Z 102,A -96.4282,B 24.9403,C -1.785,E1 24.9942,E2 -178.1611} C_DIS
LIN {X -1.6576,Y -99.2715,Z 102,A -94.6649,B 24.9403,C -1.7847,E1 24.9991,E2 -179.9237} C_DIS
LIN {X 0.6853,Y -99.2806,Z 102,A -93.5894,B 24.941,C -1.7747,E1 25.002,E2 -180.9755} C_DIS
Enddeposition()
LIN {X 0.6853,Y -99.2806,Z 102,A -93.5894,B 24.941,C -1.7747,E1 25.002,E2 -180.9755} C_DIS
Startdeposition()
$VEL.CP = VEL_PRINT
LIN {X -0.0111,Y -98.4247,Z 102,A -94.6466,B 24.9416,C -1.7655,E1 24.999,E2 -179.8966} C_DIS
LIN {X -2.4221,Y -98.3949,Z 102,A -95.9492,B 24.9414,C -1.769,E1 24.9954,E2 -178.6022} C_DIS
LIN {X -5.057,Y -98.2936,Z 102,A -97.4841,B 24.9414,C -1.7688,E1 24.9911,E2 -177.0666} C_DIS
LIN {X -7.2387,Y -98.1582,Z 102,A -98.9614,B 24.9419,C -1.7614,E1 24.987,E2 -175.571} C_DIS
LIN {X -10.7136,Y -97.8392,Z 102,A -101.0096,B 24.9419,C -1.761,E1 24.9813,E2 -173.5207} C_DIS
LIN {X -14.4566,Y -97.3572,Z 102,A -103.0919,B 24.9416,C -1.7655,E1 24.9755,E2 -171.4476} C_DIS
LIN {X -16.8467,Y -96.9722,Z 102,A -104.4955,B 24.9416,C -1.7662,E1 24.9717,E2 -170.0442} C_DIS
LIN {X -19.777,Y -96.4155,Z 102,A -106.2175,B 24.9415,C -1.7674,E1 24.9669,E2 -168.3232} C_DIS
LIN {X -22.9817,Y -95.7029,Z 102,A -107.9282,B 24.9409,C -1.7755,E1 24.9623,E2 -166.6296} C_DIS
LIN {X -25.3171,Y -95.1118,Z 102,A -109.4516,B 24.9411,C -1.772,E1 24.9582,E2 -165.0956} C_DIS
LIN {X -27.6379,Y -94.4635,Z 102,A -110.8827,B 24.9411,C -1.772,E1 24.9543,E2 -163.662} C_DIS
LIN {X -29.728,Y -93.8279,Z 102,A -112.1301,B 24.9411,C -1.7737,E1 24.951,E2 -162.4167} C_DIS
LIN {X -32.2291,Y -92.9973,Z 102,A -113.6672,B 24.941,C -1.7749,E1 24.9469,E2 -160.8794} C_DIS
LIN {X -34.512,Y -92.1745,Z 102,A -115.0831,B 24.9409,C -1.776,E1 24.9432,E2 -159.4634} C_DIS
LIN {X -36.9979,Y -91.2044,Z 102,A -116.7474,B 24.941,C -1.7737,E1 24.9389,E2 -157.7898} C_DIS
LIN {X -40.2157,Y -89.8322,Z 102,A -118.6536,B 24.9406,C -1.7804,E1 24.934,E2 -155.8952} C_DIS
LIN {X -42.2973,Y -88.8715,Z 102,A -120.0183,B 24.9406,C -1.7809,E1 24.9306,E2 -154.5282} C_DIS
LIN {X -44.4588,Y -87.8102,Z 102,A -121.3029,B 24.9402,C -1.7867,E1 24.9274,E2 -153.254} C_DIS
LIN {X -46.5939,Y -86.6962,Z 102,A -122.7112,B 24.9401,C -1.7883,E1 24.9239,E2 -151.8456} C_DIS
LIN {X -48.8512,Y -85.444,Z 102,A -124.2728,B 24.9401,C -1.7883,E1 24.9201,E2 -150.2795} C_DIS
LIN {X -52.0445,Y -83.5371,Z 102,A -126.2885,B 24.9395,C -1.7967,E1 24.9153,E2 -148.2775} C_DIS
LIN {X -53.6984,Y -82.4856,Z 102,A -127.7813,B 24.9402,C -1.7863,E1 24.9117,E2 -146.7551} C_DIS
LIN {X -56.1251,Y -80.852,Z 102,A -129.4622,B 24.94,C -1.7898,E1 24.9079,E2 -145.077} C_DIS
LIN {X -59.0085,Y -78.7724,Z 102,A -131.4813,B 24.9396,C -1.7951,E1 24.9033,E2 -143.0634} C_DIS
LIN {X -61.4977,Y -76.847,Z 102,A -133.497,B 24.9398,C -1.7921,E1 24.8989,E2 -141.0331} C_DIS
LIN {X -64.2785,Y -74.5365,Z 102,A -135.5253,B 24.9394,C -1.7987,E1 24.8946,E2 -139.0128} C_DIS
LIN {X -66.6332,Y -72.4369,Z 102,A -137.3697,B 24.9391,C -1.8022,E1 24.8908,E2 -137.1691} C_DIS
LIN {X -69.1701,Y -70.0183,Z 102,A -139.397,B 24.9388,C -1.8069,E1 24.8867,E2 -135.1445} C_DIS
LIN {X -71.284,Y -67.8677,Z 102,A -141.3536,B 24.939,C -1.8038,E1 24.8829,E2 -133.1723} C_DIS
LIN {X -73.9181,Y -64.9869,Z 102,A -143.4601,B 24.9383,C -1.8145,E1 24.879,E2 -131.082} C_DIS
LIN {X -76.1146,Y -62.4015,Z 102,A -145.5207,B 24.9382,C -1.8162,E1 24.8753,E2 -129.0159} C_DIS
LIN {X -78.3343,Y -59.5916,Z 102,A -147.5188,B 24.9376,C -1.8242,E1 24.8719,E2 -127.0272} C_DIS
LIN {X -79.9016,Y -57.4712,Z 102,A -148.9602,B 24.9372,C -1.8311,E1 24.8695,E2 -125.5953} C_DIS
LIN {X -81.2141,Y -55.6021,Z 102,A -150.3608,B 24.9371,C -1.8321,E1 24.8673,E2 -124.1901} C_DIS
LIN {X -82.8505,Y -53.1306,Z 102,A -152.1292,B 24.9369,C -1.8351,E1 24.8646,E2 -122.42} C_DIS
LIN {X -84.5932,Y -50.3104,Z 102,A -153.7927,B 24.9359,C -1.8491,E1 24.8622,E2 -120.7813} C_DIS
LIN {X -85.9146,Y -48.0183,Z 102,A -155.6137,B 24.9363,C -1.8439,E1 24.8597,E2 -118.9384} C_DIS
LIN {X -87.3685,Y -45.3231,Z 102,A -157.3159,B 24.9357,C -1.8514,E1 24.8574,E2 -117.2451} C_DIS
LIN {X -88.4523,Y -43.1698,Z 102,A -158.8308,B 24.9357,C -1.8516,E1 24.8555,E2 -115.7225} C_DIS
LIN {X -89.4916,Y -40.9716,Z 102,A -160.252,B 24.9355,C -1.8554,E1 24.8539,E2 -114.3027} C_DIS
LIN {X -90.6817,Y -38.2609,Z 102,A -161.7522,B 24.9346,C -1.8678,E1 24.8522,E2 -112.8236} C_DIS
LIN {X -91.8245,Y -35.4355,Z 102,A -163.6785,B 24.9346,C -1.8678,E1 24.8502,E2 -110.8868} C_DIS
LIN {X -92.836,Y -32.6889,Z 102,A -165.2806,B 24.934,C -1.8763,E1 24.8487,E2 -109.2957} C_DIS
LIN {X -93.5279,Y -30.6552,Z 102,A -166.5246,B 24.9337,C -1.8802,E1 24.8476,E2 -108.054} C_DIS
LIN {X -94.1867,Y -28.571,Z 102,A -167.9277,B 24.9337,C -1.8797,E1 24.8464,E2 -106.6416} C_DIS
LIN {X -94.8584,Y -26.255,Z 102,A -169.4851,B 24.9338,C -1.8789,E1 24.8453,E2 -105.0733} C_DIS
LIN {X -95.6534,Y -23.1843,Z 102,A -171.3694,B 24.9335,C -1.8834,E1 24.844,E2 -103.1887} C_DIS
LIN {X -96.2914,Y -20.3812,Z 102,A -172.8838,B 24.9328,C -1.8938,E1 24.8431,E2 -101.6901} C_DIS
LIN {X -96.8017,Y -17.7948,Z 102,A -174.3093,B 24.9322,C -1.9021,E1 24.8423,E2 -100.2761} C_DIS
LIN {X -97.2599,Y -15.0856,Z 102,A -176.1332,B 24.9323,C -1.8998,E1 24.8415,E2 -98.4359} C_DIS
LIN {X -97.7133,Y -11.8031,Z 102,A -177.9814,B 24.9317,C -1.9086,E1 24.8408,E2 -96.5974} C_DIS
LIN {X -97.9518,Y -9.6363,Z 102,A -179.3611,B 24.9317,C -1.909,E1 24.8404,E2 -95.2104} C_DIS
LIN {X -98.2035,Y -6.5692,Z 102,A 178.8465,B 24.9313,C -1.9147,E1 24.8401,E2 -93.421} C_DIS
LIN {X -98.3645,Y -3.4122,Z 102,A 177.1948,B 24.9304,C -1.9267,E1 24.8399,E2 -91.788} C_DIS
LIN {X -98.4169,Y -1.233,Z 102,A 175.7746,B 24.9304,C -1.9258,E1 24.8398,E2 -90.3572} C_DIS
LIN {X -98.4139,Y 1.3972,Z 102,A 174.3054,B 24.93,C -1.9328,E1 24.8398,E2 -88.8957} C_DIS
LIN {X -98.3581,Y 3.6214,Z 102,A 172.8561,B 24.93,C -1.9319,E1 24.8399,E2 -87.4356} C_DIS
LIN {X -98.157,Y 7.2537,Z 102,A 170.7234,B 24.9296,C -1.9383,E1 24.8403,E2 -85.3052} C_DIS
LIN {X -97.95,Y 9.6549,Z 102,A 169.4122,B 24.929,C -1.9458,E1 24.8407,E2 -84.0041} C_DIS
LIN {X -97.6315,Y 12.4576,Z 102,A 167.836,B 24.9285,C -1.9532,E1 24.8412,E2 -82.4362} C_DIS
LIN {X -97.1387,Y 15.8524,Z 102,A 165.8646,B 24.9279,C -1.9605,E1 24.842,E2 -80.4704} C_DIS
LIN {X -96.7214,Y 18.226,Z 102,A 164.2963,B 24.928,C -1.9596,E1 24.8428,E2 -78.8906} C_DIS
LIN {X -96.2912,Y 20.3821,Z 102,A 163.0412,B 24.9276,C -1.9645,E1 24.8435,E2 -77.6397} C_DIS
LIN {X -95.7071,Y 22.9645,Z 102,A 161.6147,B 24.927,C -1.9731,E1 24.8444,E2 -76.2255} C_DIS
LIN {X -95.1158,Y 25.3023,Z 102,A 160.0796,B 24.927,C -1.9733,E1 24.8454,E2 -74.6818} C_DIS
LIN {X -94.4281,Y 27.7572,Z 102,A 158.5885,B 24.9267,C -1.9777,E1 24.8466,E2 -73.1928} C_DIS
LIN {X -93.8015,Y 29.8096,Z 102,A 157.3407,B 24.9264,C -1.9817,E1 24.8476,E2 -71.9471} C_DIS
LIN {X -92.9852,Y 32.2636,Z 102,A 155.8194,B 24.9261,C -1.9859,E1 24.849,E2 -70.4272} C_DIS
LIN {X -92.1799,Y 34.4976,Z 102,A 154.4093,B 24.9258,C -1.9892,E1 24.8503,E2 -69.0172} C_DIS
LIN {X -91.3836,Y 36.5576,Z 102,A 153.1255,B 24.9255,C -1.9932,E1 24.8516,E2 -67.7357} C_DIS
LIN {X -90.4608,Y 38.7849,Z 102,A 151.6102,B 24.9255,C -1.9938,E1 24.8533,E2 -66.2134} C_DIS
LIN {X -89.4837,Y 40.989,Z 102,A 150.1968,B 24.9252,C -1.9977,E1 24.8549,E2 -64.8016} C_DIS
LIN {X -88.3304,Y 43.4156,Z 102,A 148.7275,B 24.9246,C -2.0055,E1 24.8567,E2 -63.343} C_DIS
LIN {X -87.3505,Y 45.3573,Z 102,A 147.3525,B 24.9246,C -2.0057,E1 24.8585,E2 -61.961} C_DIS
LIN {X -86.2174,Y 47.476,Z 102,A 145.9433,B 24.9243,C -2.0094,E1 24.8603,E2 -60.5533} C_DIS
LIN {X -84.9176,Y 49.7615,Z 102,A 144.6256,B 24.9234,C -2.0208,E1 24.8621,E2 -59.2559} C_DIS
LIN {X -83.6563,Y 51.8538,Z 102,A 143.2114,B 24.9231,C -2.0251,E1 24.8642,E2 -57.8448} C_DIS
LIN {X -82.5094,Y 53.6622,Z 102,A 141.7214,B 24.9234,C -2.0206,E1 24.8665,E2 -56.3364} C_DIS
LIN {X -81.16,Y 55.682,Z 102,A 140.1455,B 24.9235,C -2.0192,E1 24.869,E2 -54.7493} C_DIS
LIN {X -78.9809,Y 58.7309,Z 102,A 138.0314,B 24.9229,C -2.0274,E1 24.8724,E2 -52.6444} C_DIS
LIN {X -76.8362,Y 61.5111,Z 102,A 135.9292,B 24.9227,C -2.0309,E1 24.8761,E2 -50.5407} C_DIS
LIN {X -74.5272,Y 64.2894,Z 102,A 133.8115,B 24.9223,C -2.0358,E1 24.8799,E2 -48.4251} C_DIS
LIN {X -72.1176,Y 66.9812,Z 102,A 131.6945,B 24.9219,C -2.0407,E1 24.8839,E2 -46.3102} C_DIS
LIN {X -69.5876,Y 69.6059,Z 102,A 129.5659,B 24.9215,C -2.0456,E1 24.888,E2 -44.1844} C_DIS
LIN {X -66.9869,Y 72.1123,Z 102,A 127.4496,B 24.9212,C -2.0501,E1 24.8923,E2 -42.0701} C_DIS
LIN {X -64.2958,Y 74.5216,Z 102,A 125.3375,B 24.9208,C -2.0546,E1 24.8967,E2 -39.9603} C_DIS
LIN {X -61.7936,Y 76.6072,Z 102,A 123.5096,B 24.9203,C -2.061,E1 24.9007,E2 -38.1409} C_DIS
LIN {X -59.3629,Y 78.5062,Z 102,A 121.8485,B 24.9197,C -2.0693,E1 24.9043,E2 -36.4934} C_DIS
LIN {X -57.4403,Y 79.9237,Z 102,A 120.4503,B 24.9195,C -2.0719,E1 24.9075,E2 -35.0965} C_DIS
LIN {X -55.6644,Y 81.172,Z 102,A 119.0798,B 24.9195,C -2.0708,E1 24.9106,E2 -33.7188} C_DIS
LIN {X -53.482,Y 82.625,Z 102,A 117.7661,B 24.9188,C -2.081,E1 24.9137,E2 -32.4249} C_DIS
LIN {X -51.4206,Y 83.9233,Z 102,A 116.3406,B 24.9186,C -2.0834,E1 24.917,E2 -31.0006} C_DIS
LIN {X -49.5471,Y 85.0441,Z 102,A 114.8438,B 24.919,C -2.078,E1 24.9207,E2 -29.4865} C_DIS
LIN {X -47.4507,Y 86.2314,Z 102,A 113.4354,B 24.9188,C -2.0802,E1 24.9241,E2 -28.0793} C_DIS
LIN {X -45.0609,Y 87.5024,Z 102,A 112.1159,B 24.918,C -2.0916,E1 24.9273,E2 -26.7832} C_DIS
LIN {X -43.1731,Y 88.4507,Z 102,A 110.62,B 24.9185,C -2.0845,E1 24.9311,E2 -25.2664} C_DIS
Enddeposition()
END
